KUKA KRL program: MyProgram_201().src

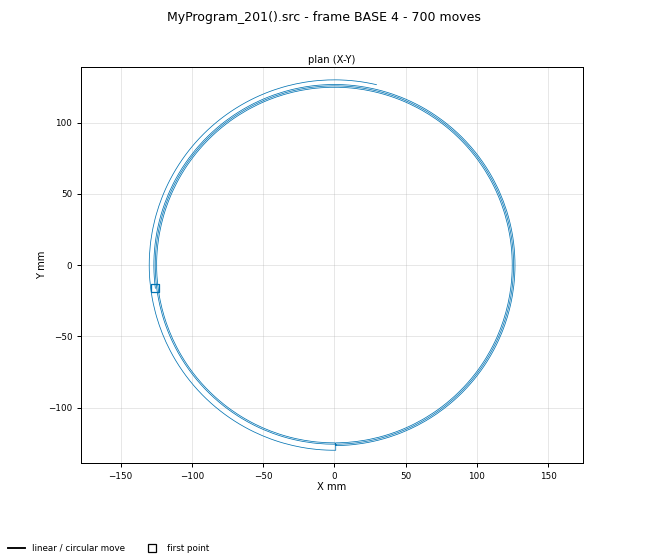
[picture p0: tool path of MyProgram_201().src in frame BASE 4, 700 of 700 moves have a stored position in this frame; points joined in program order, loops and branches not executed]
&ACCESS RVP
&REL 1
&PARAM TEMPLATE = C:\KRC\Roboter\Template\vorgabe
&PARAM EDITMASK = *
DEF MyProgram_201()
; ---- Setting reference (Base) ----
$BASE = BASE_DATA[4]

; --------------------------
; ---- Setting tool (TCP) ----
$TOOL = TOOL_DATA[3]
; --------------------------

$VEL.CP = VEL_APROX_PRINT
Startdeposition()
$VEL.CP = VEL_PRINT
LIN {X -125.6198,Y -16.3,Z 144,A -176.0579,B 23.3517,C -1.2096,E1 23.2223,E2 262.9437} C_DIS
LIN {X -126.0896,Y -12.1409,Z 144,A -177.9619,B 23.3515,C -1.2152,E1 23.2217,E2 264.8457} C_DIS
LIN {X -126.3878,Y -8.5224,Z 144,A -179.6727,B 23.3514,C -1.2176,E1 23.2214,E2 266.5617} C_DIS
LIN {X -126.5802,Y -4.8461,Z 144,A 178.7289,B 23.351,C -1.2257,E1 23.2212,E2 268.1497} C_DIS
LIN {X -126.6703,Y -1.0023,Z 144,A 177.0039,B 23.3506,C -1.2319,E1 23.2211,E2 269.8702} C_DIS
LIN {X -126.6432,Y 2.8281,Z 144,A 175.1115,B 23.3507,C -1.2309,E1 23.2211,E2 271.7776} C_DIS
LIN {X -126.4965,Y 6.6909,Z 144,A 173.3723,B 23.3504,C -1.2369,E1 23.2214,E2 273.5127} C_DIS
LIN {X -126.2226,Y 10.6706,Z 144,A 171.6302,B 23.35,C -1.2454,E1 23.2218,E2 275.2447} C_DIS
LIN {X -125.8208,Y 14.6708,Z 144,A 169.7416,B 23.3498,C -1.2483,E1 23.2223,E2 277.138} C_DIS
LIN {X -125.28,Y 18.7432,Z 144,A 167.8361,B 23.3496,C -1.2523,E1 23.2231,E2 279.0456} C_DIS
LIN {X -124.6746,Y 22.4103,Z 144,A 166.2415,B 23.3492,C -1.2614,E1 23.2238,E2 280.6274} C_DIS
LIN {X -123.8824,Y 26.4422,Z 144,A 164.0896,B 23.3495,C -1.2551,E1 23.2251,E2 282.809} C_DIS
LIN {X -122.8112,Y 31.0384,Z 144,A 162.2249,B 23.3486,C -1.2732,E1 23.2263,E2 284.6396} C_DIS
LIN {X -121.8435,Y 34.6469,Z 144,A 159.9894,B 23.3494,C -1.2558,E1 23.228,E2 286.9331} C_DIS
LIN {X -120.6189,Y 38.6913,Z 144,A 158.5603,B 23.3481,C -1.2819,E1 23.2291,E2 288.305} C_DIS
LIN {X -119.0709,Y 43.2217,Z 144,A 156.4748,B 23.3476,C -1.2919,E1 23.231,E2 290.3777} C_DIS
LIN {X -117.9603,Y 46.1668,Z 144,A 155.028,B 23.3474,C -1.2954,E1 23.2325,E2 291.8245} C_DIS
LIN {X -116.7964,Y 49.0362,Z 144,A 153.2106,B 23.3481,C -1.2823,E1 23.2345,E2 293.686} C_DIS
LIN {X -115.419,Y 52.1955,Z 144,A 151.7283,B 23.3477,C -1.2902,E1 23.2362,E2 295.1571} C_DIS
LIN {X -113.1115,Y 57.0256,Z 144,A 149.2606,B 23.3474,C -1.2954,E1 23.2392,E2 297.6257} C_DIS
LIN {X -111.6267,Y 59.8811,Z 144,A 147.8797,B 23.347,C -1.3028,E1 23.241,E2 298.9958} C_DIS
LIN {X -109.2886,Y 64.0498,Z 144,A 145.8278,B 23.3464,C -1.3137,E1 23.2439,E2 301.0317} C_DIS
LIN {X -106.917,Y 67.9358,Z 144,A 143.7293,B 23.3462,C -1.3179,E1 23.247,E2 303.1311} C_DIS
LIN {X -104.5298,Y 71.5536,Z 144,A 141.7868,B 23.3459,C -1.3241,E1 23.25,E2 305.0683} C_DIS
LIN {X -102.0291,Y 75.0763,Z 144,A 139.8415,B 23.3456,C -1.3298,E1 23.2531,E2 307.0093} C_DIS
LIN {X -97.7758,Y 80.538,Z 144,A 136.8601,B 23.3448,C -1.3444,E1 23.2583,E2 309.9688} C_DIS
LIN {X -95.6486,Y 83.0531,Z 144,A 135.1365,B 23.3451,C -1.3384,E1 23.2614,E2 311.7162} C_DIS
LIN {X -91.6576,Y 87.4372,Z 144,A 132.8632,B 23.3438,C -1.3624,E1 23.2656,E2 313.9395} C_DIS
LIN {X -88.5294,Y 90.6034,Z 144,A 130.4673,B 23.3444,C -1.351,E1 23.2704,E2 316.3752} C_DIS
LIN {X -85.4652,Y 93.4997,Z 144,A 128.2304,B 23.3449,C -1.3415,E1 23.2751,E2 318.646} C_DIS
LIN {X -82.7854,Y 95.88,Z 144,A 126.8175,B 23.3443,C -1.354,E1 23.278,E2 320.0333} C_DIS
LIN {X -79.5981,Y 98.542,Z 144,A 125.0127,B 23.3439,C -1.3612,E1 23.2819,E2 321.8271} C_DIS
LIN {X -76.158,Y 101.2243,Z 144,A 123.1143,B 23.3435,C -1.3686,E1 23.2861,E2 323.7143} C_DIS
LIN {X -70.9814,Y 104.9191,Z 144,A 120.1884,B 23.3433,C -1.3722,E1 23.2928,E2 326.6418} C_DIS
LIN {X -67.4074,Y 107.2505,Z 144,A 118.1775,B 23.3433,C -1.3724,E1 23.2975,E2 328.6591} C_DIS
LIN {X -63.7154,Y 109.4843,Z 144,A 116.2997,B 23.3429,C -1.3791,E1 23.302,E2 330.5261} C_DIS
LIN {X -60.2851,Y 111.4101,Z 144,A 114.4465,B 23.3429,C -1.379,E1 23.3065,E2 332.3853} C_DIS
LIN {X -56.9815,Y 113.134,Z 144,A 112.7261,B 23.3429,C -1.3802,E1 23.3108,E2 334.1076} C_DIS
LIN {X -52.7308,Y 115.1763,Z 144,A 110.7397,B 23.3423,C -1.3899,E1 23.3158,E2 336.075} C_DIS
LIN {X -49.6659,Y 116.5317,Z 144,A 109.2183,B 23.3422,C -1.3918,E1 23.3197,E2 337.5953} C_DIS
LIN {X -46.4891,Y 117.8349,Z 144,A 107.0676,B 23.3435,C -1.3681,E1 23.3254,E2 339.8112} C_DIS
LIN {X -42.2554,Y 119.4193,Z 144,A 105.3156,B 23.3426,C -1.3833,E1 23.3299,E2 341.5284} C_DIS
LIN {X -35.1581,Y 121.6966,Z 144,A 102.0862,B 23.3421,C -1.3933,E1 23.3385,E2 344.7386} C_DIS
LIN {X -30.6403,Y 122.9122,Z 144,A 100.1076,B 23.3416,C -1.4014,E1 23.3438,E2 346.6997} C_DIS
LIN {X -27.0358,Y 123.7543,Z 144,A 98.3688,B 23.3416,C -1.4001,E1 23.3485,E2 348.4443} C_DIS
LIN {X -23.779,Y 124.4208,Z 144,A 96.8918,B 23.3416,C -1.4025,E1 23.3526,E2 349.9172} C_DIS
LIN {X -19.8742,Y 125.1049,Z 144,A 94.9819,B 23.3418,C -1.3986,E1 23.3579,E2 351.8388} C_DIS
LIN {X -15.5594,Y 125.7148,Z 144,A 93.0348,B 23.3417,C -1.4008,E1 23.3633,E2 353.7819} C_DIS
LIN {X -11.7071,Y 126.1313,Z 144,A 90.9218,B 23.3425,C -1.3858,E1 23.3692,E2 355.9341} C_DIS
LIN {X -7.8333,Y 126.4304,Z 144,A 89.507,B 23.3416,C -1.4016,E1 23.3731,E2 357.3093} C_DIS
LIN {X -3.5316,Y 126.6237,Z 144,A 87.6883,B 23.3412,C -1.408,E1 23.3781,E2 359.1124} C_DIS
LIN {X 0.2429,Y 126.6735,Z 144,A 85.6174,B 23.3422,C -1.3921,E1 23.384,E2 361.2235} C_DIS
LIN {X 3.5494,Y 126.6232,Z 144,A 84.81,B 23.3404,C -1.4231,E1 23.386,E2 361.9523} C_DIS
LIN {X 5.9066,Y 126.5359,Z 144,A 83.2679,B 23.3416,C -1.4017,E1 23.3905,E2 363.5479} C_DIS
LIN {X 10.1935,Y 126.2629,Z 144,A 81.4048,B 23.3414,C -1.4052,E1 23.3956,E2 365.4013} C_DIS
LIN {X 13.9971,Y 125.8979,Z 144,A 79.6067,B 23.3416,C -1.4018,E1 23.4007,E2 367.2067} C_DIS
LIN {X 18.4024,Y 125.3298,Z 144,A 77.6752,B 23.3414,C -1.4048,E1 23.406,E2 369.1289} C_DIS
LIN {X 22.234,Y 124.7062,Z 144,A 75.9188,B 23.3414,C -1.4041,E1 23.4108,E2 370.8849} C_DIS
LIN {X 26.3969,Y 123.8922,Z 144,A 74.0065,B 23.3415,C -1.4035,E1 23.416,E2 372.7962} C_DIS
LIN {X 29.8566,Y 123.1039,Z 144,A 72.4577,B 23.3415,C -1.4052,E1 23.4202,E2 374.3385} C_DIS
LIN {X 33.465,Y 122.174,Z 144,A 70.6308,B 23.3418,C -1.3976,E1 23.4252,E2 376.1815} C_DIS
LIN {X 37.2836,Y 121.0616,Z 144,A 68.5449,B 23.3427,C -1.3832,E1 23.4309,E2 378.2997} C_DIS
LIN {X 40.9331,Y 119.8781,Z 144,A 67.3255,B 23.3414,C -1.4053,E1 23.4339,E2 379.4609} C_DIS
LIN {X 46.9072,Y 117.6684,Z 144,A 64.503,B 23.3414,C -1.4052,E1 23.4413,E2 382.2771} C_DIS
LIN {X 50.4597,Y 116.1885,Z 144,A 62.6584,B 23.3418,C -1.3985,E1 23.4461,E2 384.1339} C_DIS
LIN {X 53.5436,Y 114.8005,Z 144,A 60.934,B 23.3424,C -1.3876,E1 23.4505,E2 385.8809} C_DIS
LIN {X 58.0942,Y 112.5675,Z 144,A 58.8505,B 23.342,C -1.3944,E1 23.4557,E2 387.9413} C_DIS
LIN {X 60.6229,Y 111.2261,Z 144,A 57.3893,B 23.3426,C -1.3849,E1 23.4593,E2 389.4219} C_DIS
LIN {X 63.5642,Y 109.5718,Z 144,A 55.9184,B 23.3426,C -1.3852,E1 23.4628,E2 390.8872} C_DIS
LIN {X 67.2338,Y 107.3598,Z 144,A 53.9488,B 23.3428,C -1.3808,E1 23.4675,E2 392.8613} C_DIS
LIN {X 70.8573,Y 105.0027,Z 144,A 51.8125,B 23.3434,C -1.3691,E1 23.4726,E2 395.0192} C_DIS
LIN {X 73.5099,Y 103.1635,Z 144,A 50.8381,B 23.3423,C -1.3894,E1 23.4747,E2 395.939} C_DIS
LIN {X 76.0074,Y 101.338,Z 144,A 49.1263,B 23.3433,C -1.3722,E1 23.4786,E2 397.6875} C_DIS
LIN {X 79.7456,Y 98.423,Z 144,A 47.0444,B 23.3433,C -1.3711,E1 23.4831,E2 399.7637} C_DIS
LIN {X 83.033,Y 95.6661,Z 144,A 45.111,B 23.3435,C -1.3676,E1 23.4872,E2 401.6977} C_DIS
LIN {X 86.1377,Y 92.8802,Z 144,A 43.2356,B 23.3437,C -1.3643,E1 23.4911,E2 403.5732} C_DIS
LIN {X 89.0952,Y 90.0471,Z 144,A 41.3667,B 23.344,C -1.3596,E1 23.4949,E2 405.4457} C_DIS
LIN {X 92.215,Y 86.8491,Z 144,A 39.2479,B 23.3445,C -1.3505,E1 23.499,E2 407.5774} C_DIS
LIN {X 95.66,Y 83.04,Z 144,A 37.0516,B 23.3445,C -1.3512,E1 23.503,E2 409.7614} C_DIS
LIN {X 98.5681,Y 79.5657,Z 144,A 34.8905,B 23.345,C -1.341,E1 23.5069,E2 411.9373} C_DIS
LIN {X 100.9397,Y 76.5352,Z 144,A 33.2696,B 23.3449,C -1.3424,E1 23.5096,E2 413.5464} C_DIS
LIN {X 103.7767,Y 72.6422,Z 144,A 31.1105,B 23.3451,C -1.3379,E1 23.5131,E2 415.7056} C_DIS
LIN {X 106.2024,Y 69.0465,Z 144,A 29.1812,B 23.3453,C -1.3343,E1 23.5161,E2 417.6334} C_DIS
LIN {X 108.9015,Y 64.7054,Z 144,A 26.6855,B 23.3461,C -1.3194,E1 23.5197,E2 420.1529} C_DIS
LIN {X 111.4774,Y 60.16,Z 144,A 24.4951,B 23.3461,C -1.3212,E1 23.5227,E2 422.3265} C_DIS
LIN {X 113.137,Y 56.9755,Z 144,A 23.0738,B 23.3458,C -1.3264,E1 23.5245,E2 423.7263} C_DIS
LIN {X 114.3455,Y 54.507,Z 144,A 21.7849,B 23.3461,C -1.3207,E1 23.526,E2 425.0222} C_DIS
LIN {X 115.7212,Y 51.5224,Z 144,A 20.2942,B 23.3463,C -1.3163,E1 23.5278,E2 426.5154} C_DIS
LIN {X 118.532,Y 44.6783,Z 144,A 17.2084,B 23.3462,C -1.3191,E1 23.531,E2 429.5757} C_DIS
LIN {X 120.9837,Y 37.5382,Z 144,A 13.7256,B 23.3469,C -1.3054,E1 23.5341,E2 433.0715} C_DIS
LIN {X 122.1821,Y 33.436,Z 144,A 11.5325,B 23.3479,C -1.2869,E1 23.5358,E2 435.2977} C_DIS
LIN {X 123.1385,Y 29.7129,Z 144,A 9.9468,B 23.3477,C -1.2889,E1 23.5369,E2 436.8683} C_DIS
LIN {X 123.9757,Y 26.01,Z 144,A 8.1829,B 23.3481,C -1.2813,E1 23.5379,E2 438.6404} C_DIS
LIN {X 124.6529,Y 22.5315,Z 144,A 6.636,B 23.3483,C -1.279,E1 23.5387,E2 440.1833} C_DIS
LIN {X 125.2127,Y 19.1782,Z 144,A 5.1321,B 23.3484,C -1.2758,E1 23.5394,E2 441.6857} C_DIS
LIN {X 125.7472,Y 15.2874,Z 144,A 3.322,B 23.3488,C -1.2685,E1 23.5401,E2 443.5026} C_DIS
LIN {X 126.1487,Y 11.5259,Z 144,A 1.4148,B 23.3496,C -1.2534,E1 23.5406,E2 445.4354} C_DIS
LIN {X 126.4634,Y 7.2985,Z 144,A -0.699,B 23.3504,C -1.2377,E1 23.541,E2 447.5752} C_DIS
LIN {X 126.6257,Y 3.4602,Z 144,A -2.0172,B 23.3496,C -1.2525,E1 23.541,E2 448.8477} C_DIS
LIN {X 126.6741,Y -0.4435,Z 144,A -4.1027,B 23.3507,C -1.2311,E1 23.541,E2 450.9733} C_DIS
LIN {X 126.6143,Y -3.867,Z 144,A -5.4652,B 23.3505,C -1.2352,E1 23.541,E2 452.3169} C_DIS
LIN {X 126.4545,Y -7.4424,Z 144,A -6.8931,B 23.3503,C -1.2393,E1 23.5408,E2 453.7254} C_DIS
LIN {X 126.205,Y -10.8793,Z 144,A -8.4102,B 23.3504,C -1.2363,E1 23.5404,E2 455.2405} C_DIS
LIN {X 125.8638,Y -14.3081,Z 144,A -10.5466,B 23.3521,C -1.203,E1 23.5397,E2 457.4466} C_DIS
LIN {X 125.2715,Y -18.7982,Z 144,A -11.9025,B 23.3507,C -1.2301,E1 23.5392,E2 458.7259} C_DIS
LIN {X 124.8446,Y -21.4515,Z 144,A -13.3029,B 23.3514,C -1.2172,E1 23.5386,E2 460.15} C_DIS
LIN {X 124.1494,Y -25.1576,Z 144,A -14.8753,B 23.3514,C -1.2182,E1 23.5377,E2 461.7098} C_DIS
LIN {X 123.4731,Y -28.2905,Z 144,A -16.3225,B 23.3515,C -1.2137,E1 23.5369,E2 463.1592} C_DIS
LIN {X 122.6734,Y -31.581,Z 144,A -17.9398,B 23.352,C -1.2046,E1 23.5358,E2 464.7893} C_DIS
LIN {X 121.313,Y -36.4621,Z 144,A -20.3518,B 23.3526,C -1.1914,E1 23.5339,E2 467.2194} C_DIS
LIN {X 119.6559,Y -41.574,Z 144,A -22.5939,B 23.3526,C -1.193,E1 23.5319,E2 469.4439} C_DIS
LIN {X 118.4529,Y -44.8894,Z 144,A -24.0956,B 23.3526,C -1.1926,E1 23.5305,E2 470.9375} C_DIS
LIN {X 117.2414,Y -47.9665,Z 144,A -26.4217,B 23.3547,C -1.1477,E1 23.5279,E2 473.3624} C_DIS
LIN {X 115.0168,Y -53.0757,Z 144,A -28.1096,B 23.3532,C -1.1804,E1 23.5261,E2 474.9584} C_DIS
LIN {X 113.536,Y -56.1738,Z 144,A -29.6697,B 23.3534,C -1.1754,E1 23.5242,E2 476.522} C_DIS
LIN {X 111.7463,Y -59.6594,Z 144,A -31.5581,B 23.3539,C -1.1645,E1 23.5217,E2 478.4272} C_DIS
LIN {X 109.5491,Y -63.6034,Z 144,A -33.578,B 23.3541,C -1.1596,E1 23.5189,E2 480.4481} C_DIS
LIN {X 106.9185,Y -67.933,Z 144,A -35.6562,B 23.354,C -1.1634,E1 23.5159,E2 482.5054} C_DIS
LIN {X 105.1316,Y -70.6674,Z 144,A -37.6491,B 23.3553,C -1.1342,E1 23.5127,E2 484.5607} C_DIS
LIN {X 102.9247,Y -73.8438,Z 144,A -38.9435,B 23.3545,C -1.1514,E1 23.5107,E2 485.8052} C_DIS
LIN {X 100.1435,Y -77.5733,Z 144,A -41.3778,B 23.3555,C -1.1297,E1 23.5065,E2 488.2814} C_DIS
LIN {X 98.0196,Y -80.2405,Z 144,A -43.2162,B 23.3564,C -1.1114,E1 23.5032,E2 490.1566} C_DIS
LIN {X 94.8372,Y -83.9778,Z 144,A -44.5715,B 23.3547,C -1.1474,E1 23.5009,E2 491.415} C_DIS
LIN {X 92.9285,Y -86.0858,Z 144,A -46.7033,B 23.3567,C -1.1034,E1 23.4966,E2 493.6472} C_DIS
LIN {X 89.5202,Y -89.6248,Z 144,A -48.8548,B 23.3568,C -1.1013,E1 23.4924,E2 495.794} C_DIS
LIN {X 86.2046,Y -92.8179,Z 144,A -50.2021,B 23.3554,C -1.1317,E1 23.4898,E2 497.0592} C_DIS
LIN {X 83.859,Y -94.9423,Z 144,A -52.375,B 23.3572,C -1.0928,E1 23.4851,E2 499.3204} C_DIS
LIN {X 80.2421,Y -98.0183,Z 144,A -54.5894,B 23.3575,C -1.0848,E1 23.4803,E2 501.5457} C_DIS
LIN {X 76.2072,Y -101.1872,Z 144,A -56.044,B 23.3559,C -1.1212,E1 23.4773,E2 502.9032} C_DIS
LIN {X 71.3958,Y -104.6377,Z 144,A -59.0041,B 23.3568,C -1.1022,E1 23.4705,E2 505.9001} C_DIS
LIN {X 67.4922,Y -107.197,Z 144,A -61.0279,B 23.3568,C -1.1022,E1 23.4657,E2 507.9165} C_DIS
LIN {X 63.8251,Y -109.4206,Z 144,A -62.9374,B 23.3568,C -1.1001,E1 23.4611,E2 509.825} C_DIS
LIN {X 58.3747,Y -112.4216,Z 144,A -65.6581,B 23.3568,C -1.0997,E1 23.4545,E2 512.5384} C_DIS
LIN {X 55.9472,Y -113.6477,Z 144,A -66.9097,B 23.357,C -1.0967,E1 23.4513,E2 513.7939} C_DIS
LIN {X 52.9996,Y -115.052,Z 144,A -69.3957,B 23.3592,C -1.047,E1 23.4448,E2 516.3982} C_DIS
LIN {X 46.9171,Y -117.6644,Z 144,A -71.3464,B 23.3572,C -1.0915,E1 23.44,E2 518.2319} C_DIS
LIN {X 43.9008,Y -118.8222,Z 144,A -73.6629,B 23.3591,C -1.0495,E1 23.4337,E2 520.6489} C_DIS
LIN {X 38.4967,Y -120.6811,Z 144,A -75.0613,B 23.3568,C -1.1019,E1 23.4303,E2 521.9125} C_DIS
LIN {X 34.3658,Y -121.9221,Z 144,A -77.3662,B 23.3576,C -1.083,E1 23.424,E2 524.2606} C_DIS
LIN {X 31.1656,Y -122.7789,Z 144,A -78.8431,B 23.3576,C -1.0825,E1 23.42,E2 525.7365} C_DIS
LIN {X 27.8817,Y -123.5665,Z 144,A -80.5186,B 23.358,C -1.0741,E1 23.4154,E2 527.4305} C_DIS
LIN {X 23.6583,Y -124.4438,Z 144,A -82.3488,B 23.3578,C -1.0781,E1 23.4104,E2 529.2482} C_DIS
LIN {X 19.6454,Y -125.1403,Z 144,A -84.5124,B 23.3585,C -1.0618,E1 23.4044,E2 531.4506} C_DIS
LIN {X 16.3427,Y -125.6142,Z 144,A -85.6833,B 23.3579,C -1.0765,E1 23.4012,E2 532.5834} C_DIS
LIN {X 13.4015,Y -125.962,Z 144,A -86.9789,B 23.3579,C -1.0778,E1 23.3977,E2 533.8748} C_DIS
LIN {X 9.8751,Y -126.289,Z 144,A -89.1079,B 23.3589,C -1.0527,E1 23.3916,E2 536.0658} C_DIS
LIN {X 5.8614,Y -126.5377,Z 144,A -90.569,B 23.3583,C -1.0684,E1 23.3876,E2 537.4867} C_DIS
LIN {X 0.8935,Y -126.6682,Z 144,A -91.828,B 23.3563,C -1.1136,E1 23.3844,E2 538.6315} C_DIS
Enddeposition()
LIN {X 0.8935,Y -126.6682,Z 144,A -91.828,B 23.3563,C -1.1136,E1 23.3844,E2 538.6315} C_DIS
Startdeposition()
$VEL.CP = VEL_PRINT
LIN {X 1.3973,Y -125.7042,Z 144,A -91.3697,B 22.5452,C -0.9874,E1 22.5695,E2 538.3914} C_DIS
LIN {X 4.7103,Y -125.622,Z 144,A -89.8294,B 22.5452,C -0.9893,E1 22.5738,E2 536.8467} C_DIS
LIN {X 9.6558,Y -125.3397,Z 144,A -87.6305,B 22.5452,C -0.9876,E1 22.5799,E2 534.6534} C_DIS
LIN {X 13.3287,Y -125.0015,Z 144,A -86.0596,B 22.5454,C -0.9836,E1 22.5842,E2 533.0942} C_DIS
LIN {X 17.0917,Y -124.5446,Z 144,A -84.1177,B 22.5449,C -0.9943,E1 22.5897,E2 531.1261} C_DIS
LIN {X 21.777,Y -123.8099,Z 144,A -82.1653,B 22.5453,C -0.9864,E1 22.595,E2 529.1964} C_DIS
LIN {X 25.3135,Y -123.1351,Z 144,A -80.4656,B 22.5451,C -0.9905,E1 22.5996,E2 527.4884} C_DIS
LIN {X 29.4259,Y -122.2173,Z 144,A -78.6487,B 22.5452,C -0.9876,E1 22.6046,E2 525.682} C_DIS
LIN {X 32.6566,Y -121.3943,Z 144,A -77.1248,B 22.5452,C -0.9893,E1 22.6087,E2 524.1561} C_DIS
LIN {X 37.8213,Y -119.8862,Z 144,A -74.5204,B 22.5447,C -0.999,E1 22.6157,E2 521.5317} C_DIS
LIN {X 44.3034,Y -117.6443,Z 144,A -71.5515,B 22.5449,C -0.9958,E1 22.6235,E2 518.578} C_DIS
LIN {X 48.1574,Y -116.1201,Z 144,A -69.8944,B 22.5452,C -0.9878,E1 22.6277,E2 516.9458} C_DIS
LIN {X 50.0092,Y -115.3343,Z 144,A -68.364,B 22.544,C -1.0174,E1 22.6318,E2 515.3426} C_DIS
LIN {X 53.5193,Y -113.7503,Z 144,A -66.9131,B 22.5444,C -1.006,E1 22.6354,E2 513.9255} C_DIS
LIN {X 56.4487,Y -112.3248,Z 144,A -65.3839,B 22.5443,C -1.0105,E1 22.6392,E2 512.3894} C_DIS
LIN {X 60.5754,Y -110.1551,Z 144,A -63.3016,B 22.5442,C -1.0121,E1 22.6443,E2 510.3094} C_DIS
LIN {X 64.4835,Y -107.9133,Z 144,A -61.4039,B 22.5443,C -1.0086,E1 22.6489,E2 508.4273} C_DIS
LIN {X 67.5262,Y -106.0362,Z 144,A -59.7903,B 22.5443,C -1.0109,E1 22.6527,E2 506.8135} C_DIS
LIN {X 70.7564,Y -103.9088,Z 144,A -58.0963,B 22.5443,C -1.0112,E1 22.6566,E2 505.1252} C_DIS
LIN {X 73.8837,Y -101.7084,Z 144,A -56.2124,B 22.5438,C -1.0213,E1 22.6609,E2 503.2224} C_DIS
LIN {X 77.115,Y -99.2807,Z 144,A -54.3822,B 22.5436,C -1.0247,E1 22.665,E2 501.391} C_DIS
LIN {X 79.4373,Y -97.4326,Z 144,A -53.0769,B 22.5436,C -1.0254,E1 22.6678,E2 500.0892} C_DIS
LIN {X 83.6912,Y -93.804,Z 144,A -50.6755,B 22.5436,C -1.0243,E1 22.6729,E2 497.7013} C_DIS
LIN {X 87.0109,Y -90.732,Z 144,A -48.3133,B 22.5428,C -1.0432,E1 22.6778,E2 495.3008} C_DIS
LIN {X 90.6624,Y -87.0837,Z 144,A -45.932,B 22.5425,C -1.0503,E1 22.6824,E2 492.9126} C_DIS
LIN {X 93.5791,Y -83.9425,Z 144,A -43.4883,B 22.5413,C -1.0784,E1 22.6871,E2 490.4081} C_DIS
LIN {X 97.0736,Y -79.8764,Z 144,A -41.7141,B 22.5424,C -1.053,E1 22.6901,E2 488.7089} C_DIS
LIN {X 100.5173,Y -75.4965,Z 144,A -39.2558,B 22.5423,C -1.056,E1 22.6943,E2 486.2561} C_DIS
LIN {X 102.6274,Y -72.6018,Z 144,A -37.53,B 22.5419,C -1.0648,E1 22.6972,E2 484.5167} C_DIS
LIN {X 104.4261,Y -69.9902,Z 144,A -36.0169,B 22.5416,C -1.0721,E1 22.6995,E2 482.9932} C_DIS
LIN {X 106.5615,Y -66.6943,Z 144,A -34.3365,B 22.5416,C -1.0719,E1 22.702,E2 481.3226} C_DIS
LIN {X 108.8374,Y -62.9111,Z 144,A -32.4123,B 22.5415,C -1.0735,E1 22.7048,E2 479.4054} C_DIS
LIN {X 110.8877,Y -59.2233,Z 144,A -30.3838,B 22.541,C -1.0841,E1 22.7075,E2 477.3613} C_DIS
LIN {X 112.6381,Y -55.8176,Z 144,A -29.0173,B 22.5416,C -1.0714,E1 22.7092,E2 476.036} C_DIS
LIN {X 113.7558,Y -53.5079,Z 144,A -27.6617,B 22.541,C -1.0837,E1 22.7108,E2 474.6567} C_DIS
LIN {X 115.4559,Y -49.7279,Z 144,A -25.7582,B 22.5407,C -1.0901,E1 22.713,E2 472.7483} C_DIS
LIN {X 116.9827,Y -46.0242,Z 144,A -23.872,B 22.5403,C -1.0985,E1 22.7149,E2 470.8519} C_DIS
LIN {X 118.0398,Y -43.243,Z 144,A -22.5259,B 22.5402,C -1.1022,E1 22.7163,E2 469.5047} C_DIS
LIN {X 119.5913,Y -38.7445,Z 144,A -20.5598,B 22.5403,C -1.0993,E1 22.718,E2 467.5584} C_DIS
LIN {X 121.2999,Y -33.0105,Z 144,A -17.6404,B 22.5395,C -1.117,E1 22.7203,E2 464.612} C_DIS
LIN {X 122.25,Y -29.2905,Z 144,A -16.0088,B 22.5395,C -1.117,E1 22.7214,E2 462.9912} C_DIS
LIN {X 123.0731,Y -25.6183,Z 144,A -14.3435,B 22.5393,C -1.12,E1 22.7224,E2 461.3287} C_DIS
LIN {X 123.7616,Y -22.0466,Z 144,A -12.6352,B 22.539,C -1.1277,E1 22.7232,E2 459.6117} C_DIS
LIN {X 124.4349,Y -17.8596,Z 144,A -10.6377,B 22.5385,C -1.137,E1 22.7241,E2 457.6034} C_DIS
LIN {X 124.996,Y -13.3799,Z 144,A -8.7163,B 22.5385,C -1.137,E1 22.7247,E2 455.6943} C_DIS
LIN {X 125.3442,Y -9.5941,Z 144,A -7.1161,B 22.5385,C -1.1364,E1 22.7251,E2 454.1066} C_DIS
LIN {X 125.5162,Y -7.0136,Z 144,A -5.6321,B 22.5377,C -1.1547,E1 22.7253,E2 452.5851} C_DIS
LIN {X 125.6659,Y -3.337,Z 144,A -4.1352,B 22.5378,C -1.1515,E1 22.7255,E2 451.1064} C_DIS
LIN {X 125.7109,Y 0.4944,Z 144,A -2.2888,B 22.5373,C -1.1618,E1 22.7255,E2 449.2455} C_DIS
LIN {X 125.6122,Y 4.9598,Z 144,A -0.3445,B 22.5373,C -1.164,E1 22.7253,E2 447.3085} C_DIS
LIN {X 125.3828,Y 9.0647,Z 144,A 1.5442,B 22.5369,C -1.1707,E1 22.725,E2 445.415} C_DIS
LIN {X 125.0498,Y 12.8794,Z 144,A 3.3043,B 22.5366,C -1.177,E1 22.7245,E2 443.6504} C_DIS
LIN {X 124.5826,Y 16.8046,Z 144,A 5.0302,B 22.5365,C -1.1791,E1 22.7239,E2 441.9305} C_DIS
LIN {X 124.0343,Y 20.4578,Z 144,A 6.6901,B 22.5363,C -1.1833,E1 22.7232,E2 440.2707} C_DIS
LIN {X 123.3637,Y 24.1809,Z 144,A 8.4722,B 22.5359,C -1.1914,E1 22.7222,E2 438.4793} C_DIS
LIN {X 122.6818,Y 27.4311,Z 144,A 9.9685,B 22.5357,C -1.1952,E1 22.7214,E2 436.9827} C_DIS
LIN {X 121.8425,Y 30.9412,Z 144,A 11.5191,B 22.5357,C -1.1959,E1 22.7203,E2 435.4405} C_DIS
LIN {X 120.8108,Y 34.7569,Z 144,A 13.3945,B 22.5352,C -1.2048,E1 22.7189,E2 433.554} C_DIS
LIN {X 119.1746,Y 40.0056,Z 144,A 15.8059,B 22.535,C -1.2079,E1 22.7169,E2 431.1499} C_DIS
LIN {X 117.9546,Y 43.4749,Z 144,A 17.5608,B 22.5346,C -1.2165,E1 22.7152,E2 429.3837} C_DIS
LIN {X 116.6595,Y 46.8349,Z 144,A 19.4072,B 22.5339,C -1.231,E1 22.7133,E2 427.5112} C_DIS
LIN {X 115.4102,Y 49.8337,Z 144,A 20.5484,B 22.5345,C -1.2193,E1 22.712,E2 426.4074} C_DIS
LIN {X 113.8888,Y 53.2213,Z 144,A 22.2347,B 22.5342,C -1.2238,E1 22.7101,E2 424.7197} C_DIS
LIN {X 112.4489,Y 56.2012,Z 144,A 23.6966,B 22.5342,C -1.2258,E1 22.7083,E2 423.2613} C_DIS
LIN {X 110.4675,Y 60.003,Z 144,A 25.6015,B 22.534,C -1.2289,E1 22.7058,E2 421.3597} C_DIS
LIN {X 106.7236,Y 66.4338,Z 144,A 29.1203,B 22.5332,C -1.2438,E1 22.7008,E2 417.8224} C_DIS
LIN {X 104.517,Y 69.854,Z 144,A 30.973,B 22.5329,C -1.2485,E1 22.6979,E2 415.968} C_DIS
LIN {X 102.3735,Y 72.9595,Z 144,A 32.854,B 22.5323,C -1.2604,E1 22.6949,E2 414.0665} C_DIS
LIN {X 99.8538,Y 76.3714,Z 144,A 35.3234,B 22.5307,C -1.2902,E1 22.6906,E2 411.5328} C_DIS
LIN {X 96.3505,Y 80.7463,Z 144,A 37.1616,B 22.5322,C -1.2627,E1 22.6874,E2 409.7753} C_DIS
LIN {X 93.4225,Y 84.1172,Z 144,A 39.1811,B 22.532,C -1.2667,E1 22.6837,E2 407.7558} C_DIS
LIN {X 90.4829,Y 87.2713,Z 144,A 41.153,B 22.5317,C -1.2713,E1 22.6799,E2 405.7814} C_DIS
LIN {X 87.5036,Y 90.258,Z 144,A 43.0584,B 22.5316,C -1.2746,E1 22.6761,E2 403.8765} C_DIS
LIN {X 84.1876,Y 93.3594,Z 144,A 45.1451,B 22.5313,C -1.2796,E1 22.6718,E2 401.7863} C_DIS
LIN {X 80.894,Y 96.2265,Z 144,A 47.0415,B 22.5313,C -1.2792,E1 22.6678,E2 399.8992} C_DIS
LIN {X 77.7947,Y 98.7491,Z 144,A 48.7644,B 22.5313,C -1.2781,E1 22.6641,E2 398.1865} C_DIS
LIN {X 74.6266,Y 101.1648,Z 144,A 50.59,B 22.5312,C -1.2818,E1 22.66,E2 396.3587} C_DIS
LIN {X 68.4588,Y 105.4361,Z 144,A 54.0629,B 22.5307,C -1.2898,E1 22.652,E2 392.878} C_DIS
LIN {X 65.0458,Y 107.5752,Z 144,A 55.9453,B 22.5305,C -1.2948,E1 22.6475,E2 390.9895} C_DIS
LIN {X 61.7684,Y 109.4901,Z 144,A 57.9194,B 22.5297,C -1.3083,E1 22.6426,E2 388.9868} C_DIS
LIN {X 58.9101,Y 111.053,Z 144,A 58.9352,B 22.5308,C -1.2891,E1 22.6403,E2 388.0241} C_DIS
LIN {X 53.407,Y 113.8029,Z 144,A 61.8058,B 22.5304,C -1.2956,E1 22.6331,E2 385.1453} C_DIS
LIN {X 50.1312,Y 115.2816,Z 144,A 63.447,B 22.5304,C -1.2976,E1 22.6289,E2 383.5033} C_DIS
LIN {X 47.4059,Y 116.4293,Z 144,A 64.6842,B 22.5305,C -1.2941,E1 22.6257,E2 382.2785} C_DIS
LIN {X 45.0897,Y 117.346,Z 144,A 66.1802,B 22.5296,C -1.3114,E1 22.6217,E2 380.7413} C_DIS
LIN {X 40.9801,Y 118.8428,Z 144,A 67.9313,B 22.5301,C -1.3024,E1 22.6172,E2 379.0176} C_DIS
LIN {X 38.2253,Y 119.7571,Z 144,A 69.4464,B 22.5295,C -1.312,E1 22.6131,E2 377.4806} C_DIS
LIN {X 33.614,Y 121.1326,Z 144,A 71.5799,B 22.5295,C -1.3109,E1 22.6074,E2 375.3539} C_DIS
LIN {X 29.5738,Y 122.1817,Z 144,A 73.3621,B 22.5298,C -1.3068,E1 22.6026,E2 373.5856} C_DIS
LIN {X 26.7358,Y 122.8341,Z 144,A 74.6078,B 22.53,C -1.3039,E1 22.5992,E2 372.3493} C_DIS
LIN {X 24.26,Y 123.3486,Z 144,A 76.0118,B 22.5293,C -1.3155,E1 22.5953,E2 370.9169} C_DIS
LIN {X 20.2227,Y 124.0736,Z 144,A 77.8245,B 22.5294,C -1.3137,E1 22.5903,E2 369.1112} C_DIS
LIN {X 16.6715,Y 124.6001,Z 144,A 79.4068,B 22.5295,C -1.3117,E1 22.5859,E2 367.5354} C_DIS
LIN {X 12.7934,Y 125.0591,Z 144,A 81.1548,B 22.5295,C -1.3106,E1 22.5811,E2 365.7916} C_DIS
LIN {X 9.6513,Y 125.34,Z 144,A 82.6613,B 22.5295,C -1.3138,E1 22.5769,E2 364.2779} C_DIS
LIN {X 5.8843,Y 125.573,Z 144,A 84.4407,B 22.5293,C -1.3164,E1 22.5719,E2 362.4924} C_DIS
LIN {X 2.548,Y 125.6852,Z 144,A 85.9635,B 22.5293,C -1.3163,E1 22.5677,E2 360.9701} C_DIS
LIN {X -1.588,Y 125.7011,Z 144,A 87.7905,B 22.5294,C -1.3134,E1 22.5626,E2 359.1507} C_DIS
LIN {X -5.8581,Y 125.5743,Z 144,A 89.6412,B 22.5297,C -1.3086,E1 22.5575,E2 357.3121} C_DIS
LIN {X -9.2502,Y 125.3693,Z 144,A 91.2103,B 22.5297,C -1.3089,E1 22.5531,E2 355.7415} C_DIS
LIN {X -12.6393,Y 125.0746,Z 144,A 92.8985,B 22.5294,C -1.3141,E1 22.5483,E2 354.0388} C_DIS
LIN {X -17.0334,Y 124.5526,Z 144,A 94.8862,B 22.5295,C -1.3117,E1 22.5429,E2 352.0558} C_DIS
LIN {X -20.8143,Y 123.9749,Z 144,A 96.5383,B 22.5298,C -1.3066,E1 22.5383,E2 350.4153} C_DIS
LIN {X -24.7961,Y 123.2404,Z 144,A 98.1445,B 22.5305,C -1.295,E1 22.534,E2 348.8375} C_DIS
LIN {X -27.7971,Y 122.5982,Z 144,A 99.7818,B 22.53,C -1.3039,E1 22.5295,E2 347.1745} C_DIS
LIN {X -30.7189,Y 121.8989,Z 144,A 101.5782,B 22.529,C -1.3209,E1 22.5245,E2 345.3309} C_DIS
LIN {X -34.5541,Y 120.8697,Z 144,A 102.8963,B 22.5303,C -1.298,E1 22.5211,E2 344.0704} C_DIS
LIN {X -41.9598,Y 118.5024,Z 144,A 106.5271,B 22.5303,C -1.2975,E1 22.5115,E2 340.4334} C_DIS
LIN {X -45.6938,Y 117.1111,Z 144,A 108.2688,B 22.5306,C -1.292,E1 22.5069,E2 338.7019} C_DIS
LIN {X -48.0993,Y 116.1444,Z 144,A 109.4942,B 22.5306,C -1.2922,E1 22.5037,E2 337.4729} C_DIS
LIN {X -51.1847,Y 114.8175,Z 144,A 110.9613,B 22.5309,C -1.2874,E1 22.5,E2 336.0146} C_DIS
LIN {X -53.5421,Y 113.7394,Z 144,A 112.3507,B 22.5305,C -1.2943,E1 22.4964,E2 334.6033} C_DIS
LIN {X -56.9349,Y 112.0773,Z 144,A 113.9501,B 22.5309,C -1.2864,E1 22.4925,E2 333.0196} C_DIS
LIN {X -59.9517,Y 110.4955,Z 144,A 115.5264,B 22.531,C -1.2848,E1 22.4886,E2 331.4427} C_DIS
LIN {X -62.9409,Y 108.8201,Z 144,A 117.1463,B 22.531,C -1.2845,E1 22.4847,E2 329.8181} C_DIS
LIN {X -66.1966,Y 106.8712,Z 144,A 118.9254,B 22.531,C -1.2835,E1 22.4804,E2 328.0357} C_DIS
LIN {X -69.4711,Y 104.7726,Z 144,A 120.721,B 22.5312,C -1.281,E1 22.4762,E2 326.2399} C_DIS
LIN {X -73.3963,Y 102.0612,Z 144,A 122.9053,B 22.5314,C -1.2771,E1 22.4712,E2 324.0574} C_DIS
LIN {X -76.7078,Y 99.5964,Z 144,A 124.8137,B 22.5316,C -1.2743,E1 22.467,E2 322.1485} C_DIS
LIN {X -80.0002,Y 96.9711,Z 144,A 126.7172,B 22.5318,C -1.2695,E1 22.4629,E2 320.2496} C_DIS
LIN {X -82.7086,Y 94.6714,Z 144,A 128.3509,B 22.532,C -1.2665,E1 22.4594,E2 318.6166} C_DIS
LIN {X -85.9752,Y 91.7158,Z 144,A 130.3928,B 22.5322,C -1.2633,E1 22.4552,E2 316.5739} C_DIS
LIN {X -89.1602,Y 88.6219,Z 144,A 132.3209,B 22.5326,C -1.2546,E1 22.4514,E2 314.6596} C_DIS
LIN {X -91.5259,Y 86.1765,Z 144,A 133.9755,B 22.5326,C -1.255,E1 22.4482,E2 312.9957} C_DIS
LIN {X -94.5489,Y 82.849,Z 144,A 136.0275,B 22.5329,C -1.25,E1 22.4444,E2 310.9466} C_DIS
LIN {X -97.4805,Y 79.3787,Z 144,A 137.983,B 22.5334,C -1.24,E1 22.441,E2 309.0073} C_DIS
LIN {X -100.2604,Y 75.8369,Z 144,A 140.1506,B 22.5334,C -1.2392,E1 22.4372,E2 306.83} C_DIS
LIN {X -102.7076,Y 72.4882,Z 144,A 142.0685,B 22.5336,C -1.2353,E1 22.4341,E2 304.9121} C_DIS
LIN {X -105.2217,Y 68.7891,Z 144,A 144.1516,B 22.5338,C -1.2314,E1 22.4309,E2 302.8273} C_DIS
LIN {X -107.4248,Y 65.2946,Z 144,A 145.988,B 22.5342,C -1.2242,E1 22.4282,E2 300.9993} C_DIS
LIN {X -109.347,Y 62.0218,Z 144,A 147.5096,B 22.5349,C -1.2108,E1 22.4261,E2 299.504} C_DIS
LIN {X -111.9896,Y 57.1071,Z 144,A 150.2199,B 22.5349,C -1.2102,E1 22.4226,E2 296.7793} C_DIS
LIN {X -113.591,Y 53.8527,Z 144,A 152.5902,B 22.5337,C -1.2345,E1 22.4196,E2 294.3307} C_DIS
LIN {X -115.73,Y 49.0914,Z 144,A 154.2621,B 22.5355,C -1.1984,E1 22.4179,E2 292.743} C_DIS
LIN {X -116.8988,Y 46.2401,Z 144,A 155.8427,B 22.5354,C -1.2013,E1 22.4162,E2 291.145} C_DIS
LIN {X -118.2627,Y 42.6247,Z 144,A 157.535,B 22.5358,C -1.1931,E1 22.4146,E2 289.4634} C_DIS
LIN {X -119.7087,Y 38.377,Z 144,A 159.634,B 22.536,C -1.189,E1 22.4127,E2 287.3618} C_DIS
LIN {X -120.9621,Y 34.2238,Z 144,A 161.539,B 22.5365,C -1.1798,E1 22.4113,E2 285.4684} C_DIS
LIN {X -121.7696,Y 31.2286,Z 144,A 162.784,B 22.537,C -1.1686,E1 22.4104,E2 284.2449} C_DIS
LIN {X -122.4845,Y 28.295,Z 144,A 164.1298,B 22.5373,C -1.163,E1 22.4095,E2 282.9049} C_DIS
LIN {X -123.043,Y 25.7663,Z 144,A 165.8093,B 22.5365,C -1.1794,E1 22.4085,E2 281.1712} C_DIS
LIN {X -123.9653,Y 20.8718,Z 144,A 167.7007,B 22.5376,C -1.1569,E1 22.4076,E2 279.3263} C_DIS
LIN {X -124.4315,Y 17.8833,Z 144,A 169.2086,B 22.5376,C -1.1577,E1 22.407,E2 277.8062} C_DIS
LIN {X -124.946,Y 13.8445,Z 144,A 171.0221,B 22.5379,C -1.15,E1 22.4064,E2 276.0007} C_DIS
LIN {X -125.2603,Y 10.6244,Z 144,A 172.563,B 22.538,C -1.148,E1 22.406,E2 274.4548} C_DIS
LIN {X -125.5343,Y 6.6543,Z 144,A 174.4112,B 22.5382,C -1.1435,E1 22.4057,E2 272.6057} C_DIS
LIN {X -125.6838,Y 2.6278,Z 144,A 176.2903,B 22.5384,C -1.1394,E1 22.4055,E2 270.725} C_DIS
LIN {X -125.7065,Y -1.1296,Z 144,A 178.0855,B 22.5385,C -1.1372,E1 22.4055,E2 268.9232} C_DIS
LIN {X -125.6053,Y -5.137,Z 144,A 179.8881,B 22.5389,C -1.1304,E1 22.4057,E2 267.1263} C_DIS
LIN {X -125.413,Y -8.6522,Z 144,A -178.6267,B 22.5393,C -1.1204,E1 22.406,E2 265.6572} C_DIS
LIN {X -125.1003,Y -12.3711,Z 144,A -176.7514,B 22.5393,C -1.1221,E1 22.4064,E2 263.7649} C_DIS
LIN {X -124.6415,Y -16.3554,Z 144,A -175.0218,B 22.5397,C -1.1123,E1 22.407,E2 262.0493} C_DIS
LIN {X -124.0525,Y -20.3488,Z 144,A -173.2265,B 22.5401,C -1.1048,E1 22.4078,E2 260.2619} C_DIS
LIN {X -123.4772,Y -23.5874,Z 144,A -171.8662,B 22.5405,C -1.0945,E1 22.4085,E2 258.9196} C_DIS
LIN {X -122.4488,Y -28.4512,Z 144,A -169.2579,B 22.5402,C -1.1013,E1 22.41,E2 256.276} C_DIS
LIN {X -120.6353,Y -35.3564,Z 144,A -166.1216,B 22.5409,C -1.0866,E1 22.4123,E2 253.1579} C_DIS
LIN {X -119.435,Y -39.2235,Z 144,A -164.1564,B 22.5409,C -1.086,E1 22.414,E2 251.1818} C_DIS
LIN {X -118.4461,Y -42.1159,Z 144,A -162.796,B 22.5412,C -1.0805,E1 22.4153,E2 249.8271} C_DIS
LIN {X -117.2159,Y -45.4243,Z 144,A -161.2592,B 22.5415,C -1.0729,E1 22.4168,E2 248.3005} C_DIS
LIN {X -116.0214,Y -48.3937,Z 144,A -159.7551,B 22.5416,C -1.0705,E1 22.4184,E2 246.7933} C_DIS
LIN {X -114.6413,Y -51.5787,Z 144,A -158.2161,B 22.5419,C -1.0642,E1 22.4201,E2 245.2613} C_DIS
LIN {X -113.3524,Y -54.3523,Z 144,A -156.7544,B 22.5419,C -1.0631,E1 22.4218,E2 243.7936} C_DIS
LIN {X -111.5604,Y -57.9438,Z 144,A -154.8529,B 22.5421,C -1.0609,E1 22.4243,E2 241.8863} C_DIS
LIN {X -109.5033,Y -61.745,Z 144,A -152.8502,B 22.5422,C -1.0569,E1 22.427,E2 239.8822} C_DIS
LIN {X -107.3306,Y -65.4494,Z 144,A -150.8548,B 22.5424,C -1.0533,E1 22.4298,E2 237.8848} C_DIS
LIN {X -104.7434,Y -69.5148,Z 144,A -148.619,B 22.5426,C -1.0493,E1 22.4332,E2 235.6469} C_DIS
LIN {X -102.1315,Y -73.2979,Z 144,A -146.542,B 22.5428,C -1.0433,E1 22.4366,E2 233.5743} C_DIS
LIN {X -99.4314,Y -76.9207,Z 144,A -144.4475,B 22.543,C -1.0397,E1 22.4401,E2 231.4778} C_DIS
LIN {X -96.5398,Y -80.5207,Z 144,A -142.3317,B 22.5432,C -1.0352,E1 22.4439,E2 229.3628} C_DIS
LIN {X -93.5469,Y -83.9784,Z 144,A -140.3033,B 22.5435,C -1.0282,E1 22.4476,E2 227.3426} C_DIS
LIN {X -90.6491,Y -87.0989,Z 144,A -138.3121,B 22.5435,C -1.026,E1 22.4514,E2 225.3474} C_DIS
LIN {X -87.7943,Y -89.9757,Z 144,A -136.4441,B 22.5437,C -1.023,E1 22.4551,E2 223.4785} C_DIS
LIN {X -84.662,Y -92.9289,Z 144,A -134.4788,B 22.5439,C -1.0191,E1 22.4591,E2 221.5143} C_DIS
LIN {X -81.4152,Y -95.7859,Z 144,A -132.702,B 22.5444,C -1.0071,E1 22.4628,E2 219.7612} C_DIS
LIN {X -78.1,Y -98.508,Z 144,A -130.6301,B 22.5444,C -1.0084,E1 22.4674,E2 217.6772} C_DIS
LIN {X -74.8635,Y -100.9896,Z 144,A -128.2574,B 22.5435,C -1.027,E1 22.4728,E2 215.2463} C_DIS
LIN {X -71.3984,Y -103.4686,Z 144,A -126.7074,B 22.5444,C -1.007,E1 22.4763,E2 213.7426} C_DIS
LIN {X -67.7176,Y -105.9137,Z 144,A -124.8621,B 22.5448,C -0.9967,E1 22.4805,E2 211.9177} C_DIS
LIN {X -64.8026,Y -107.7223,Z 144,A -122.9919,B 22.5444,C -1.0074,E1 22.4851,E2 210.0129} C_DIS
LIN {X -60.6058,Y -110.1382,Z 144,A -121.1441,B 22.5452,C -0.989,E1 22.4895,E2 208.2073} C_DIS
LIN {X -56.2275,Y -112.4359,Z 144,A -118.666,B 22.5449,C -0.9957,E1 22.4957,E2 205.7041} C_DIS
LIN {X -52.9512,Y -114.0137,Z 144,A -117.0944,B 22.5451,C -0.9901,E1 22.4996,E2 204.1427} C_DIS
LIN {X -49.7493,Y -115.4467,Z 144,A -115.4714,B 22.5451,C -0.9893,E1 22.5038,E2 202.5173} C_DIS
LIN {X -45.6775,Y -117.1175,Z 144,A -113.7812,B 22.5458,C -0.9737,E1 22.5081,E2 200.8637} C_DIS
LIN {X -43.2432,Y -118.0397,Z 144,A -112.1574,B 22.5451,C -0.9915,E1 22.5124,E2 199.1898} C_DIS
LIN {X -38.7562,Y -119.5875,Z 144,A -110.0668,B 22.5453,C -0.9866,E1 22.5179,E2 197.1077} C_DIS
LIN {X -35.5337,Y -120.5834,Z 144,A -108.5905,B 22.5454,C -0.9828,E1 22.5219,E2 195.6383} C_DIS
LIN {X -32.3214,Y -121.4837,Z 144,A -107.0667,B 22.5454,C -0.982,E1 22.526,E2 194.1141} C_DIS
LIN {X -28.4745,Y -122.4435,Z 144,A -105.4069,B 22.5458,C -0.9745,E1 22.5304,E2 192.4712} C_DIS
LIN {X -25.2113,Y -123.1559,Z 144,A -103.7563,B 22.5456,C -0.9794,E1 22.535,E2 190.8055} C_DIS
LIN {X -21.9427,Y -123.7802,Z 144,A -102.2073,B 22.5456,C -0.9803,E1 22.5392,E2 189.2525} C_DIS
LIN {X -17.7249,Y -124.4541,Z 144,A -100.3835,B 22.5458,C -0.9744,E1 22.5442,E2 187.4425} C_DIS
LIN {X -15.3658,Y -124.7683,Z 144,A -99.3374,B 22.5458,C -0.9724,E1 22.5471,E2 186.4005} C_DIS
LIN {X -12.5775,Y -125.0805,Z 144,A -97.7909,B 22.5454,C -0.9841,E1 22.5515,E2 184.8226} C_DIS
LIN {X -8.3106,Y -125.4364,Z 144,A -95.9605,B 22.5456,C -0.9787,E1 22.5566,E2 183.0055} C_DIS
LIN {X -5.8356,Y -125.5755,Z 144,A -94.6305,B 22.5452,C -0.9876,E1 22.5604,E2 181.6518} C_DIS
LIN {X -1.6894,Y -125.6994,Z 144,A -92.8902,B 22.5455,C -0.9812,E1 22.5652,E2 179.9281} C_DIS
LIN {X 0.888,Y -125.7071,Z 144,A -92.1808,B 22.5463,C -0.9608,E1 22.567,E2 179.2719} C_DIS
Enddeposition()
LIN {X 0.888,Y -125.7071,Z 144,A -92.1808,B 22.5463,C -0.9608,E1 22.567,E2 179.2719} C_DIS
Startdeposition()
$VEL.CP = VEL_PRINT
LIN {X 0.2524,Y -124.7479,Z 144,A -92.4528,B 21.6328,C -0.8169,E1 21.6473,E2 179.8151} C_DIS
LIN {X -2.8004,Y -124.7177,Z 144,A -93.8116,B 21.6328,C -0.8185,E1 21.6435,E2 181.1697} C_DIS
LIN {X -5.8687,Y -124.6098,Z 144,A -95.3337,B 21.6329,C -0.8138,E1 21.6392,E2 182.7051} C_DIS
LIN {X -8.918,Y -124.4282,Z 144,A -96.719,B 21.6329,C -0.8145,E1 21.6353,E2 184.0889} C_DIS
LIN {X -11.9747,Y -124.1712,Z 144,A -98.1094,B 21.6329,C -0.8154,E1 21.6315,E2 185.4777} C_DIS
LIN {X -15.2704,Y -123.81,Z 144,A -99.586,B 21.6329,C -0.8176,E1 21.6274,E2 186.9496} C_DIS
LIN {X -18.2991,Y -123.3995,Z 144,A -100.9842,B 21.6328,C -0.8181,E1 21.6235,E2 188.3477} C_DIS
LIN {X -21.0776,Y -122.9548,Z 144,A -102.3448,B 21.6328,C -0.8157,E1 21.6197,E2 189.7162} C_DIS
LIN {X -24.0877,Y -122.4013,Z 144,A -103.7803,B 21.6328,C -0.815,E1 21.6158,E2 191.1554} C_DIS
LIN {X -27.0795,Y -121.7746,Z 144,A -105.1144,B 21.6328,C -0.8186,E1 21.6122,E2 192.4818} C_DIS
LIN {X -30.8178,Y -120.8805,Z 144,A -106.9181,B 21.6328,C -0.818,E1 21.6073,E2 194.29} C_DIS
LIN {X -34.7477,Y -119.8103,Z 144,A -108.7516,B 21.6327,C -0.8208,E1 21.6024,E2 196.1193} C_DIS
LIN {X -38.3606,Y -118.7032,Z 144,A -110.6677,B 21.6329,C -0.8148,E1 21.5972,E2 198.0558} C_DIS
LIN {X -42.0313,Y -117.4532,Z 144,A -112.1555,B 21.6324,C -0.8282,E1 21.5934,E2 199.5105} C_DIS
LIN {X -44.6529,Y -116.4828,Z 144,A -113.554,B 21.6325,C -0.8247,E1 21.5897,E2 200.9218} C_DIS
LIN {X -47.7441,Y -115.2493,Z 144,A -115.0912,B 21.6325,C -0.8259,E1 21.5857,E2 202.4598} C_DIS
LIN {X -50.322,Y -114.1487,Z 144,A -116.3775,B 21.6325,C -0.8273,E1 21.5824,E2 203.7457} C_DIS
LIN {X -53.1051,Y -112.8812,Z 144,A -117.8779,B 21.6325,C -0.8251,E1 21.5786,E2 205.2567} C_DIS
LIN {X -55.6295,Y -111.6573,Z 144,A -119.1842,B 21.6325,C -0.826,E1 21.5753,E2 206.5646} C_DIS
LIN {X -58.8172,Y -110.0129,Z 144,A -120.8764,B 21.6325,C -0.8263,E1 21.5711,E2 208.2614} C_DIS
LIN {X -62.7594,Y -107.8127,Z 144,A -122.7937,B 21.6322,C -0.8354,E1 21.5665,E2 210.1604} C_DIS
LIN {X -65.2277,Y -106.3371,Z 144,A -124.1927,B 21.6322,C -0.8343,E1 21.5631,E2 211.5676} C_DIS
LIN {X -68.0304,Y -104.5663,Z 144,A -125.8027,B 21.6322,C -0.8332,E1 21.5593,E2 213.1868} C_DIS
LIN {X -71.6486,Y -102.1215,Z 144,A -127.7456,B 21.632,C -0.8389,E1 21.5549,E2 215.1216} C_DIS
LIN {X -74.3226,Y -100.192,Z 144,A -129.1995,B 21.6318,C -0.8439,E1 21.5516,E2 216.568} C_DIS
LIN {X -77.3473,Y -97.8763,Z 144,A -131.1281,B 21.632,C -0.84,E1 21.5473,E2 218.5156} C_DIS
LIN {X -80.9006,Y -94.9597,Z 144,A -133.2085,B 21.6318,C -0.8452,E1 21.5429,E2 220.5911} C_DIS
LIN {X -83.9176,Y -92.3044,Z 144,A -135.0595,B 21.6317,C -0.8486,E1 21.539,E2 222.4414} C_DIS
LIN {X -87.1252,Y -89.2834,Z 144,A -137.1298,B 21.6316,C -0.851,E1 21.5348,E2 224.5154} C_DIS
LIN {X -90.3489,Y -86.0196,Z 144,A -139.2549,B 21.6314,C -0.8548,E1 21.5307,E2 226.6408} C_DIS
LIN {X -93.3636,Y -82.7374,Z 144,A -141.3112,B 21.6313,C -0.859,E1 21.5269,E2 228.6965} C_DIS
LIN {X -96.3526,Y -79.2374,Z 144,A -143.4384,B 21.6311,C -0.8634,E1 21.523,E2 230.8232} C_DIS
LIN {X -99.286,Y -75.529,Z 144,A -145.6202,B 21.6309,C -0.8682,E1 21.5193,E2 233.0041} C_DIS
LIN {X -101.8411,Y -72.0462,Z 144,A -147.5137,B 21.6306,C -0.8765,E1 21.5162,E2 234.8855} C_DIS
LIN {X -103.4952,Y -69.6498,Z 144,A -148.8323,B 21.6304,C -0.8806,E1 21.5142,E2 236.2007} C_DIS
LIN {X -105.394,Y -66.7412,Z 144,A -150.4044,B 21.6303,C -0.8856,E1 21.5118,E2 237.7684} C_DIS
LIN {X -107.3381,Y -63.568,Z 144,A -152.2689,B 21.6303,C -0.8841,E1 21.5091,E2 239.6483} C_DIS
LIN {X -109.0083,Y -60.6589,Z 144,A -153.7998,B 21.6301,C -0.8886,E1 21.507,E2 241.1764} C_DIS
LIN {X -110.7313,Y -57.4517,Z 144,A -155.3541,B 21.6298,C -0.8977,E1 21.505,E2 242.7157} C_DIS
LIN {X -112.105,Y -54.722,Z 144,A -156.7717,B 21.6296,C -0.901,E1 21.5032,E2 244.1331} C_DIS
LIN {X -113.3721,Y -52.0448,Z 144,A -158.1603,B 21.6296,C -0.9038,E1 21.5016,E2 245.5231} C_DIS
LIN {X -114.6559,Y -49.1522,Z 144,A -159.5638,B 21.6293,C -0.9098,E1 21.5,E2 246.9192} C_DIS
LIN {X -115.7277,Y -46.5712,Z 144,A -160.9466,B 21.6293,C -0.9098,E1 21.4985,E2 248.3113} C_DIS
LIN {X -116.9316,Y -43.4612,Z 144,A -162.4448,B 21.6291,C -0.9154,E1 21.4971,E2 249.8039} C_DIS
LIN {X -117.877,Y -40.8265,Z 144,A -163.8657,B 21.6291,C -0.9141,E1 21.4957,E2 251.2379} C_DIS
LIN {X -119.301,Y -36.4564,Z 144,A -165.8387,B 21.6287,C -0.9256,E1 21.4941,E2 253.1929} C_DIS
LIN {X -120.1801,Y -33.4453,Z 144,A -167.3468,B 21.6286,C -0.9273,E1 21.4929,E2 254.7064} C_DIS
LIN {X -120.9512,Y -30.5395,Z 144,A -168.7032,B 21.6284,C -0.9325,E1 21.492,E2 256.0582} C_DIS
LIN {X -121.7122,Y -27.3526,Z 144,A -170.1618,B 21.6281,C -0.9388,E1 21.4911,E2 257.5095} C_DIS
LIN {X -122.2999,Y -24.5897,Z 144,A -171.5531,B 21.6281,C -0.9392,E1 21.4903,E2 258.9093} C_DIS
LIN {X -122.8665,Y -21.5829,Z 144,A -172.9593,B 21.6279,C -0.9435,E1 21.4896,E2 260.3135} C_DIS
LIN {X -123.4657,Y -17.8359,Z 144,A -174.7563,B 21.6278,C -0.9469,E1 21.4888,E2 262.1139} C_DIS
LIN {X -123.9605,Y -14.0034,Z 144,A -176.5073,B 21.6275,C -0.9533,E1 21.4882,E2 263.8597} C_DIS
LIN {X -124.2874,Y -10.7037,Z 144,A -177.958,B 21.6272,C -0.9609,E1 21.4878,E2 265.2999} C_DIS
LIN {X -124.5122,Y -7.6551,Z 144,A -179.56,B 21.6273,C -0.9579,E1 21.4875,E2 266.9216} C_DIS
LIN {X -124.6989,Y -3.4773,Z 144,A 178.5669,B 21.627,C -0.9657,E1 21.4873,E2 268.7864} C_DIS
LIN {X -124.7512,Y 0,Z 144,A 176.9955,B 21.6267,C -0.9717,E1 21.4873,E2 270.3526} C_DIS
LIN {X -124.7178,Y 2.7981,Z 144,A 175.6188,B 21.6267,C -0.9724,E1 21.4873,E2 271.7372} C_DIS
LIN {X -124.5975,Y 6.1146,Z 144,A 174.1544,B 21.6264,C -0.9795,E1 21.4875,E2 273.1925} C_DIS
LIN {X -124.3755,Y 9.6396,Z 144,A 172.3482,B 21.6264,C -0.9778,E1 21.4879,E2 275.0163} C_DIS
LIN {X -123.9878,Y 13.7499,Z 144,A 170.6451,B 21.6259,C -0.991,E1 21.4884,E2 276.6952} C_DIS
LIN {X -123.6144,Y 16.7829,Z 144,A 169.2327,B 21.6257,C -0.9952,E1 21.4889,E2 278.1062} C_DIS
LIN {X -123.2062,Y 19.5526,Z 144,A 167.9585,B 21.6255,C -0.9997,E1 21.4894,E2 279.377} C_DIS
LIN {X -122.7289,Y 22.3518,Z 144,A 166.5947,B 21.6255,C -1.0015,E1 21.4901,E2 280.7452} C_DIS
LIN {X -122.0399,Y 25.8519,Z 144,A 165.053,B 21.625,C -1.0103,E1 21.4909,E2 282.2736} C_DIS
LIN {X -121.4301,Y 28.5832,Z 144,A 163.5749,B 21.6252,C -1.0071,E1 21.4919,E2 283.7707} C_DIS
LIN {X -120.6276,Y 31.795,Z 144,A 162.2226,B 21.6247,C -1.0182,E1 21.4928,E2 285.1019} C_DIS
LIN {X -119.8126,Y 34.7399,Z 144,A 160.7157,B 21.6247,C -1.0187,E1 21.4939,E2 286.6179} C_DIS
LIN {X -118.9904,Y 37.4616,Z 144,A 159.3317,B 21.6247,C -1.0197,E1 21.4951,E2 288.0084} C_DIS
LIN {X -117.7586,Y 41.1681,Z 144,A 157.4776,B 21.6245,C -1.023,E1 21.4968,E2 289.866} C_DIS
LIN {X -116.4821,Y 44.6548,Z 144,A 155.7332,B 21.6243,C -1.0267,E1 21.4985,E2 291.6118} C_DIS
LIN {X -114.854,Y 48.6907,Z 144,A 153.7999,B 21.6239,C -1.0351,E1 21.5005,E2 293.5347} C_DIS
LIN {X -113.5271,Y 51.7096,Z 144,A 152.3345,B 21.6236,C -1.0415,E1 21.5022,E2 294.9922} C_DIS
LIN {X -112.1064,Y 54.7192,Z 144,A 150.8971,B 21.6233,C -1.0494,E1 21.5039,E2 296.4171} C_DIS
LIN {X -110.7366,Y 57.4417,Z 144,A 149.28,B 21.6235,C -1.0453,E1 21.506,E2 298.0557} C_DIS
LIN {X -108.6685,Y 61.2653,Z 144,A 147.3341,B 21.6231,C -1.0529,E1 21.5086,E2 299.9928} C_DIS
LIN {X -107.1334,Y 63.9115,Z 144,A 145.8689,B 21.6231,C -1.0546,E1 21.5107,E2 301.4623} C_DIS
LIN {X -104.9029,Y 67.5109,Z 144,A 143.8645,B 21.6229,C -1.0577,E1 21.5137,E2 303.4702} C_DIS
LIN {X -102.8639,Y 70.5781,Z 144,A 142.3729,B 21.6223,C -1.0699,E1 21.5159,E2 304.9371} C_DIS
LIN {X -101.1034,Y 73.0779,Z 144,A 140.8902,B 21.6223,C -1.0707,E1 21.5184,E2 306.4262} C_DIS
LIN {X -99.5146,Y 75.227,Z 144,A 139.5798,B 21.6223,C -1.0708,E1 21.5206,E2 307.7437} C_DIS
LIN {X -96.9904,Y 78.4546,Z 144,A 137.7323,B 21.622,C -1.077,E1 21.5238,E2 309.5846} C_DIS
LIN {X -94.5433,Y 81.3868,Z 144,A 135.9402,B 21.6218,C -1.08,E1 21.527,E2 311.3782} C_DIS
LIN {X -91.8324,Y 84.4337,Z 144,A 133.9744,B 21.6218,C -1.0811,E1 21.5307,E2 313.3513} C_DIS
LIN {X -88.7425,Y 87.6763,Z 144,A 131.8775,B 21.6216,C -1.0845,E1 21.5348,E2 315.4495} C_DIS
LIN {X -85.4623,Y 90.8761,Z 144,A 129.7591,B 21.6214,C -1.0889,E1 21.539,E2 317.5663} C_DIS
LIN {X -82.147,Y 93.8836,Z 144,A 127.8253,B 21.621,C -1.0982,E1 21.543,E2 319.4838} C_DIS
LIN {X -79.2339,Y 96.3554,Z 144,A 126.0585,B 21.6208,C -1.1015,E1 21.5468,E2 321.2495} C_DIS
LIN {X -76.2462,Y 98.736,Z 144,A 124.1891,B 21.6208,C -1.1007,E1 21.5509,E2 323.129} C_DIS
LIN {X -73.2919,Y 100.9482,Z 144,A 122.6253,B 21.6204,C -1.1092,E1 21.5544,E2 324.6762} C_DIS
LIN {X -70.5703,Y 102.8692,Z 144,A 121.0847,B 21.6204,C -1.1118,E1 21.5579,E2 326.216} C_DIS
LIN {X -67.4871,Y 104.9181,Z 144,A 119.2472,B 21.6204,C -1.1097,E1 21.5623,E2 328.0663} C_DIS
LIN {X -64.1345,Y 107.0005,Z 144,A 117.5608,B 21.62,C -1.1178,E1 21.5662,E2 329.7366} C_DIS
LIN {X -61.7204,Y 108.4105,Z 144,A 116.222,B 21.62,C -1.1179,E1 21.5695,E2 331.0799} C_DIS
LIN {X -59.2142,Y 109.7996,Z 144,A 114.8737,B 21.62,C -1.1188,E1 21.5728,E2 332.4302} C_DIS
LIN {X -56.3046,Y 111.3178,Z 144,A 113.3999,B 21.6198,C -1.1226,E1 21.5764,E2 333.8985} C_DIS
LIN {X -53.5596,Y 112.6641,Z 144,A 111.9867,B 21.6197,C -1.1244,E1 21.58,E2 335.311} C_DIS
LIN {X -49.86,Y 114.3499,Z 144,A 110.0267,B 21.6197,C -1.1234,E1 21.585,E2 337.2791} C_DIS
LIN {X -46.5617,Y 115.7315,Z 144,A 108.4579,B 21.6195,C -1.1286,E1 21.589,E2 338.8381} C_DIS
LIN {X -43.4579,Y 116.9329,Z 144,A 106.9958,B 21.6193,C -1.1331,E1 21.5928,E2 340.2913} C_DIS
LIN {X -40.7617,Y 117.8995,Z 144,A 105.6509,B 21.6193,C -1.1336,E1 21.5964,E2 341.6382} C_DIS
LIN {X -37.8914,Y 118.8531,Z 144,A 104.2568,B 21.6192,C -1.135,E1 21.6001,E2 343.0314} C_DIS
LIN {X -34.9883,Y 119.7398,Z 144,A 102.8589,B 21.6191,C -1.1363,E1 21.6038,E2 344.4284} C_DIS
LIN {X -31.9893,Y 120.5758,Z 144,A 101.4323,B 21.6191,C -1.1379,E1 21.6077,E2 345.8534} C_DIS
LIN {X -29.0722,Y 121.3122,Z 144,A 100.0056,B 21.6191,C -1.1373,E1 21.6115,E2 347.2838} C_DIS
LIN {X -25.8354,Y 122.0435,Z 144,A 98.5372,B 21.6189,C -1.1408,E1 21.6155,E2 348.745} C_DIS
LIN {X -23.4811,Y 122.5173,Z 144,A 97.3772,B 21.6189,C -1.1394,E1 21.6187,E2 349.9103} C_DIS
LIN {X -19.8131,Y 123.1658,Z 144,A 95.6782,B 21.6189,C -1.141,E1 21.6234,E2 351.6069} C_DIS
LIN {X -17.038,Y 123.5797,Z 144,A 94.4155,B 21.6188,C -1.1429,E1 21.6269,E2 352.8657} C_DIS
LIN {X -13.7487,Y 123.9879,Z 144,A 92.7541,B 21.619,C -1.1381,E1 21.6315,E2 354.5414} C_DIS
LIN {X -9.4196,Y 124.3916,Z 144,A 90.8117,B 21.6189,C -1.1412,E1 21.6369,E2 356.4765} C_DIS
LIN {X -6.3691,Y 124.5847,Z 144,A 89.4595,B 21.6187,C -1.1437,E1 21.6407,E2 357.8222} C_DIS
LIN {X -3.3157,Y 124.7034,Z 144,A 88.0864,B 21.6187,C -1.1453,E1 21.6445,E2 359.1911} C_DIS
LIN {X -0.2603,Y 124.7479,Z 144,A 86.6834,B 21.6187,C -1.1456,E1 21.6484,E2 360.5934} C_DIS
LIN {X 2.8086,Y 124.7175,Z 144,A 85.1585,B 21.6189,C -1.1411,E1 21.6527,E2 362.1304} C_DIS
LIN {X 5.862,Y 124.6102,Z 144,A 83.776,B 21.6189,C -1.142,E1 21.6565,E2 363.51} C_DIS
LIN {X 8.9233,Y 124.4278,Z 144,A 82.3901,B 21.6188,C -1.1428,E1 21.6604,E2 364.8928} C_DIS
LIN {X 11.9697,Y 124.1717,Z 144,A 81.0025,B 21.6188,C -1.1433,E1 21.6642,E2 366.2781} C_DIS
LIN {X 15.2654,Y 123.8106,Z 144,A 79.5268,B 21.6187,C -1.1449,E1 21.6683,E2 367.7481} C_DIS
LIN {X 18.3091,Y 123.3981,Z 144,A 78.1281,B 21.6187,C -1.145,E1 21.6722,E2 369.1452} C_DIS
LIN {X 21.0762,Y 122.9551,Z 144,A 76.7723,B 21.6188,C -1.1417,E1 21.6759,E2 370.5082} C_DIS
LIN {X 24.0829,Y 122.4022,Z 144,A 75.3413,B 21.6189,C -1.14,E1 21.6799,E2 371.9421} C_DIS
LIN {X 27.0747,Y 121.7757,Z 144,A 74.033,B 21.6187,C -1.1432,E1 21.6834,E2 373.2396} C_DIS
LIN {X 31.7974,Y 120.627,Z 144,A 71.784,B 21.6188,C -1.1412,E1 21.6895,E2 375.4901} C_DIS
LIN {X 35.5282,Y 119.5818,Z 144,A 69.8449,B 21.6192,C -1.1333,E1 21.6948,E2 377.4469} C_DIS
LIN {X 39.1363,Y 118.4493,Z 144,A 68.2135,B 21.6191,C -1.1363,E1 21.6991,E2 379.0666} C_DIS
LIN {X 43.0124,Y 117.0995,Z 144,A 66.3193,B 21.6192,C -1.1341,E1 21.704,E2 380.9619} C_DIS
LIN {X 46.0884,Y 115.9224,Z 144,A 64.8074,B 21.6192,C -1.1327,E1 21.708,E2 382.4739} C_DIS
LIN {X 49.7453,Y 114.3995,Z 144,A 62.9841,B 21.6194,C -1.1305,E1 21.7127,E2 384.2979} C_DIS
LIN {X 52.7478,Y 113.047,Z 144,A 61.4294,B 21.6196,C -1.127,E1 21.7166,E2 385.8576} C_DIS
LIN {X 55.8794,Y 111.5341,Z 144,A 59.9637,B 21.6194,C -1.1305,E1 21.7203,E2 387.3092} C_DIS
LIN {X 58.1907,Y 110.3433,Z 144,A 58.866,B 21.6193,C -1.133,E1 21.723,E2 388.3964} C_DIS
LIN {X 61.2703,Y 108.6656,Z 144,A 57.1345,B 21.6196,C -1.1256,E1 21.7272,E2 390.142} C_DIS
LIN {X 63.9163,Y 107.1305,Z 144,A 55.7751,B 21.6196,C -1.1255,E1 21.7305,E2 391.4969} C_DIS
LIN {X 66.1899,Y 105.7414,Z 144,A 54.4657,B 21.6199,C -1.12,E1 21.7336,E2 392.8163} C_DIS
LIN {X 69.3784,Y 103.6769,Z 144,A 52.8217,B 21.6199,C -1.1215,E1 21.7374,E2 394.4499} C_DIS
LIN {X 71.6566,Y 102.1159,Z 144,A 51.4996,B 21.6201,C -1.117,E1 21.7405,E2 395.7786} C_DIS
LIN {X 74.2503,Y 100.2458,Z 144,A 49.9454,B 21.6204,C -1.1108,E1 21.744,E2 397.3431} C_DIS
LIN {X 77.4542,Y 97.7915,Z 144,A 48.0953,B 21.6205,C -1.1076,E1 21.7481,E2 399.1939} C_DIS
LIN {X 80.9019,Y 94.9586,Z 144,A 46.1655,B 21.6205,C -1.1088,E1 21.7522,E2 401.1117} C_DIS
LIN {X 83.7825,Y 92.4269,Z 144,A 44.2999,B 21.6208,C -1.1008,E1 21.7561,E2 402.9902} C_DIS
LIN {X 87.1229,Y 89.2857,Z 144,A 42.2041,B 21.621,C -1.0969,E1 21.7603,E2 405.0863} C_DIS
LIN {X 90.2557,Y 86.1171,Z 144,A 40.2992,B 21.621,C -1.0986,E1 21.764,E2 406.977} C_DIS
LIN {X 92.8593,Y 83.3031,Z 144,A 38.4726,B 21.6213,C -1.0918,E1 21.7675,E2 408.8125} C_DIS
LIN {X 95.5986,Y 80.1445,Z 144,A 36.5449,B 21.6215,C -1.0871,E1 21.771,E2 410.7428} C_DIS
LIN {X 98.3612,Y 76.7297,Z 144,A 34.4938,B 21.6218,C -1.0808,E1 21.7745,E2 412.7995} C_DIS
LIN {X 100.936,Y 73.3088,Z 144,A 32.6959,B 21.6217,C -1.0833,E1 21.7775,E2 414.5804} C_DIS
LIN {X 102.8684,Y 70.5715,Z 144,A 31.2399,B 21.6217,C -1.0831,E1 21.7798,E2 416.0286} C_DIS
LIN {X 104.4249,Y 68.2483,Z 144,A 29.979,B 21.6218,C -1.0808,E1 21.7818,E2 417.2883} C_DIS
LIN {X 106.067,Y 65.6668,Z 144,A 28.4361,B 21.6223,C -1.0711,E1 21.7841,E2 418.8481} C_DIS
LIN {X 107.792,Y 62.7953,Z 144,A 27.0081,B 21.6223,C -1.0719,E1 21.7861,E2 420.2655} C_DIS
LIN {X 108.9761,Y 60.7171,Z 144,A 25.8578,B 21.6225,C -1.0667,E1 21.7877,E2 421.4229} C_DIS
LIN {X 110.5089,Y 57.8754,Z 144,A 24.3687,B 21.6227,C -1.0624,E1 21.7896,E2 422.9143} C_DIS
LIN {X 112.1086,Y 54.7148,Z 144,A 22.8061,B 21.6227,C -1.0607,E1 21.7916,E2 424.4716} C_DIS
LIN {X 113.416,Y 51.9497,Z 144,A 21.2739,B 21.6232,C -1.0512,E1 21.7934,E2 426.0199} C_DIS
LIN {X 115.1579,Y 47.9629,Z 144,A 19.4096,B 21.6232,C -1.0514,E1 21.7954,E2 427.8716} C_DIS
LIN {X 116.3904,Y 44.8907,Z 144,A 17.8991,B 21.6234,C -1.0474,E1 21.797,E2 429.383} C_DIS
LIN {X 117.6166,Y 41.5776,Z 144,A 16.0769,B 21.624,C -1.0338,E1 21.7987,E2 431.2299} C_DIS
LIN {X 118.8392,Y 37.9348,Z 144,A 14.6236,B 21.6236,C -1.0424,E1 21.8,E2 432.6504} C_DIS
LIN {X 119.7384,Y 34.9932,Z 144,A 13.1346,B 21.6239,C -1.0348,E1 21.8012,E2 434.15} C_DIS
LIN {X 120.6142,Y 31.8455,Z 144,A 11.7197,B 21.6239,C -1.034,E1 21.8022,E2 435.5573} C_DIS
LIN {X 121.2895,Y 29.1664,Z 144,A 10.3346,B 21.6244,C -1.025,E1 21.8031,E2 436.9573} C_DIS
LIN {X 122.043,Y 25.8377,Z 144,A 8.8551,B 21.6244,C -1.0241,E1 21.804,E2 438.4293} C_DIS
LIN {X 122.6404,Y 22.837,Z 144,A 7.4551,B 21.6246,C -1.02,E1 21.8048,E2 439.8307} C_DIS
LIN {X 123.0327,Y 20.6106,Z 144,A 6.3703,B 21.6249,C -1.0147,E1 21.8053,E2 440.9223} C_DIS
LIN {X 123.5791,Y 17.0424,Z 144,A 4.7721,B 21.6249,C -1.0122,E1 21.8059,E2 442.5162} C_DIS
LIN {X 123.9601,Y 14.0076,Z 144,A 3.349,B 21.6252,C -1.0069,E1 21.8064,E2 443.9436} C_DIS
LIN {X 124.2871,Y 10.7069,Z 144,A 1.8461,B 21.6254,C -1.0031,E1 21.8068,E2 445.4464} C_DIS
LIN {X 124.5627,Y 6.8067,Z 144,A -0.0922,B 21.6259,C -0.991,E1 21.8071,E2 447.4037} C_DIS
LIN {X 124.7033,Y 3.3162,Z 144,A -1.5433,B 21.6259,C -0.9928,E1 21.8073,E2 448.8399} C_DIS
LIN {X 124.7512,Y 0.0032,Z 144,A -3.2805,B 21.6265,C -0.9783,E1 21.8073,E2 450.6042} C_DIS
LIN {X 124.6627,Y -4.6003,Z 144,A -5.065,B 21.6261,C -0.9863,E1 21.8072,E2 452.3545} C_DIS
LIN {X 124.5123,Y -7.6536,Z 144,A -6.594,B 21.6265,C -0.9763,E1 21.8069,E2 453.8999} C_DIS
LIN {X 124.1719,Y -11.9674,Z 144,A -8.532,B 21.6267,C -0.9721,E1 21.8065,E2 455.8355} C_DIS
LIN {X 123.8109,Y -15.2636,Z 144,A -9.9963,B 21.6268,C -0.9699,E1 21.806,E2 457.2957} C_DIS
LIN {X 123.398,Y -18.3094,Z 144,A -11.391,B 21.627,C -0.9662,E1 21.8054,E2 458.6908} C_DIS
LIN {X 122.9556,Y -21.073,Z 144,A -12.7319,B 21.6272,C -0.9596,E1 21.8048,E2 460.0402} C_DIS
LIN {X 122.4024,Y -24.0821,Z 144,A -14.155,B 21.6275,C -0.9543,E1 21.8041,E2 461.4677} C_DIS
LIN {X 121.7758,Y -27.0738,Z 144,A -15.478,B 21.6275,C -0.9535,E1 21.8033,E2 462.7838} C_DIS
LIN {X 121.0111,Y -30.3034,Z 144,A -16.9879,B 21.6277,C -0.9494,E1 21.8023,E2 464.2945} C_DIS
LIN {X 120.3015,Y -33.0112,Z 144,A -18.3523,B 21.628,C -0.9419,E1 21.8013,E2 465.6701} C_DIS
LIN {X 119.3725,Y -36.2231,Z 144,A -19.7844,B 21.628,C -0.9417,E1 21.8002,E2 467.0929} C_DIS
LIN {X 118.4518,Y -39.1287,Z 144,A -21.1782,B 21.6282,C -0.9377,E1 21.799,E2 468.4883} C_DIS
LIN {X 117.4532,Y -42.0313,Z 144,A -22.4837,B 21.6282,C -0.938,E1 21.7978,E2 469.7844} C_DIS
LIN {X 116.655,Y -44.1998,Z 144,A -23.7127,B 21.6286,C -0.9273,E1 21.7966,E2 471.0342} C_DIS
LIN {X 115.2539,Y -47.7332,Z 144,A -25.3575,B 21.6286,C -0.9265,E1 21.7949,E2 472.6704} C_DIS
LIN {X 114.1583,Y -50.3004,Z 144,A -26.6252,B 21.6288,C -0.9233,E1 21.7934,E2 473.9387} C_DIS
LIN {X 112.6583,Y -53.5716,Z 144,A -28.3846,B 21.6291,C -0.9137,E1 21.7913,E2 475.7129} C_DIS
LIN {X 111.0985,Y -56.7355,Z 144,A -29.956,B 21.6292,C -0.9111,E1 21.7894,E2 477.2814} C_DIS
LIN {X 109.4093,Y -59.9324,Z 144,A -31.5345,B 21.6292,C -0.9099,E1 21.7873,E2 478.8534} C_DIS
LIN {X 107.7788,Y -62.8181,Z 144,A -33.0119,B 21.6294,C -0.9075,E1 21.7853,E2 480.3282} C_DIS
LIN {X 106.3424,Y -65.2191,Z 144,A -34.3746,B 21.6297,C -0.9005,E1 21.7833,E2 481.7018} C_DIS
LIN {X 104.7112,Y -67.8072,Z 144,A -35.7757,B 21.6298,C -0.8967,E1 21.7812,E2 483.1046} C_DIS
LIN {X 102.8589,Y -70.5853,Z 144,A -37.1675,B 21.6298,C -0.8988,E1 21.779,E2 484.4828} C_DIS
LIN {X 101.1014,Y -73.0806,Z 144,A -38.6868,B 21.6301,C -0.8898,E1 21.7765,E2 486.0177} C_DIS
LIN {X 98.7477,Y -76.2312,Z 144,A -40.5668,B 21.6304,C -0.8817,E1 21.7733,E2 487.9089} C_DIS
LIN {X 95.9188,Y -79.7614,Z 144,A -42.6243,B 21.6306,C -0.8772,E1 21.7697,E2 489.9674} C_DIS
LIN {X 93.4479,Y -82.6421,Z 144,A -44.2886,B 21.6306,C -0.8763,E1 21.7667,E2 491.6253} C_DIS
LIN {X 90.7899,Y -85.5537,Z 144,A -46.167,B 21.6309,C -0.8689,E1 21.7631,E2 493.5142} C_DIS
LIN {X 87.6322,Y -88.7862,Z 144,A -48.247,B 21.6311,C -0.8637,E1 21.759,E2 495.5978} C_DIS
LIN {X 84.4321,Y -91.8339,Z 144,A -50.1193,B 21.6311,C -0.8659,E1 21.7552,E2 497.4552} C_DIS
LIN {X 81.5491,Y -94.4034,Z 144,A -51.9243,B 21.6312,C -0.8605,E1 21.7514,E2 499.2663} C_DIS
LIN {X 78.5306,Y -96.9291,Z 144,A -53.8154,B 21.6315,C -0.8529,E1 21.7473,E2 501.1694} C_DIS
LIN {X 75.0019,Y -99.6845,Z 144,A -55.838,B 21.6316,C -0.8501,E1 21.7428,E2 503.191} C_DIS
LIN {X 72.0526,Y -101.8366,Z 144,A -57.4443,B 21.6316,C -0.8498,E1 21.7392,E2 504.7915} C_DIS
LIN {X 69.5113,Y -103.5881,Z 144,A -58.7862,B 21.6316,C -0.8503,E1 21.7361,E2 506.1267} C_DIS
LIN {X 66.7362,Y -105.3971,Z 144,A -60.2451,B 21.6316,C -0.8501,E1 21.7327,E2 507.5804} C_DIS
LIN {X 64.1341,Y -107.0007,Z 144,A -61.6993,B 21.6318,C -0.8454,E1 21.7292,E2 509.0421} C_DIS
LIN {X 61.7189,Y -108.4114,Z 144,A -63.0275,B 21.6319,C -0.8412,E1 21.726,E2 510.3768} C_DIS
LIN {X 58.8568,Y -109.9917,Z 144,A -64.5116,B 21.632,C -0.8394,E1 21.7223,E2 511.8608} C_DIS
LIN {X 56.317,Y -111.3115,Z 144,A -65.7734,B 21.632,C -0.8396,E1 21.7192,E2 513.1181} C_DIS
LIN {X 53.5683,Y -112.6599,Z 144,A -67.228,B 21.6322,C -0.8353,E1 21.7155,E2 514.5797} C_DIS
LIN {X 50.0233,Y -114.2793,Z 144,A -69.1461,B 21.6325,C -0.8271,E1 21.7106,E2 516.5144} C_DIS
LIN {X 46.556,Y -115.7339,Z 144,A -70.7356,B 21.6323,C -0.8306,E1 21.7065,E2 518.0902} C_DIS
LIN {X 43.055,Y -117.0838,Z 144,A -72.6298,B 21.6327,C -0.821,E1 21.7015,E2 520.0056} C_DIS
LIN {X 38.7085,Y -118.5917,Z 144,A -74.7325,B 21.6327,C -0.8189,E1 21.6959,E2 522.1092} C_DIS
LIN {X 35.0384,Y -119.7252,Z 144,A -76.3289,B 21.6326,C -0.8241,E1 21.6917,E2 523.6881} C_DIS
LIN {X 31.1491,Y -120.7964,Z 144,A -78.2724,B 21.6328,C -0.8183,E1 21.6864,E2 525.6436} C_DIS
LIN {X 27.3258,Y -121.7183,Z 144,A -79.9235,B 21.6326,C -0.8233,E1 21.682,E2 527.2786} C_DIS
LIN {X 24.5874,Y -122.3004,Z 144,A -81.2335,B 21.6326,C -0.8212,E1 21.6784,E2 528.5925} C_DIS
LIN {X 21.5827,Y -122.8666,Z 144,A -82.6258,B 21.6326,C -0.8206,E1 21.6746,E2 529.9845} C_DIS
LIN {X 18.2864,Y -123.4013,Z 144,A -84.0968,B 21.6326,C -0.8222,E1 21.6705,E2 531.4495} C_DIS
LIN {X 15.5138,Y -123.7808,Z 144,A -85.4083,B 21.6327,C -0.8202,E1 21.6669,E2 532.7649} C_DIS
LIN {X 12.4797,Y -124.1227,Z 144,A -86.9136,B 21.6329,C -0.8152,E1 21.6627,E2 534.2828} C_DIS
LIN {X 9.4366,Y -124.3903,Z 144,A -88.303,B 21.6329,C -0.8152,E1 21.6588,E2 535.6715} C_DIS
LIN {X 6.3597,Y -124.5851,Z 144,A -89.6898,B 21.6329,C -0.8158,E1 21.655,E2 537.0558} C_DIS
LIN {X 3.3061,Y -124.7036,Z 144,A -91.0682,B 21.6329,C -0.8164,E1 21.6511,E2 538.4322} C_DIS
LIN {X 0.8815,Y -124.7436,Z 144,A -91.8615,B 21.6324,C -0.8296,E1 21.649,E2 539.1896} C_DIS
Enddeposition()
LIN {X 0.9207,Y -129.9307,Z 145,A -92.7827,B 24.9662,C -1.3435,E1 25.0014,E2 539.2396} C_DIS
Startdeposition()
$VEL.CP = VEL_PRINT
LIN {X -2.2482,Y -129.9156,Z 145,A -94.5027,B 24.967,C -1.3268,E1 24.9965,E2 540.9993} C_DIS
LIN {X -5.5164,Y -129.8187,Z 145,A -95.9921,B 24.9672,C -1.3242,E1 24.9923,E2 542.4951} C_DIS
LIN {X -9.3888,Y -129.5953,Z 145,A -97.6431,B 24.967,C -1.3272,E1 24.9878,E2 544.1396} C_DIS
LIN {X -12.6486,Y -129.318,Z 145,A -99.0947,B 24.967,C -1.3268,E1 24.9837,E2 545.5927} C_DIS
LIN {X -16.9567,Y -128.8237,Z 145,A -100.9838,B 24.967,C -1.3283,E1 24.9785,E2 547.4796} C_DIS
LIN {X -20.0422,Y -128.3799,Z 145,A -102.4087,B 24.967,C -1.3261,E1 24.9745,E2 548.911} C_DIS
LIN {X -23.6437,Y -127.7678,Z 145,A -103.9695,B 24.967,C -1.3292,E1 24.9703,E2 550.4661} C_DIS
LIN {X -26.5827,Y -127.1884,Z 145,A -105.2739,B 24.9668,C -1.3306,E1 24.9667,E2 551.7687} C_DIS
LIN {X -29.2429,Y -126.6017,Z 145,A -106.5224,B 24.9669,C -1.3288,E1 24.9633,E2 553.0229} C_DIS
LIN {X -32.7218,Y -125.7494,Z 145,A -108.0816,B 24.9669,C -1.3307,E1 24.9591,E2 554.5799} C_DIS
LIN {X -35.534,Y -124.9827,Z 145,A -109.3697,B 24.9668,C -1.3315,E1 24.9556,E2 555.8683} C_DIS
LIN {X -38.2773,Y -124.169,Z 145,A -110.6285,B 24.9668,C -1.3325,E1 24.9522,E2 557.1267} C_DIS
LIN {X -41.494,Y -123.1319,Z 145,A -112.1369,B 24.9668,C -1.3329,E1 24.9482,E2 558.637} C_DIS
LIN {X -44.5442,Y -122.0617,Z 145,A -113.5399,B 24.9666,C -1.3352,E1 24.9445,E2 560.0372} C_DIS
LIN {X -47.5418,Y -120.9257,Z 145,A -114.9754,B 24.9666,C -1.3355,E1 24.9408,E2 561.4751} C_DIS
LIN {X -50.4597,Y -119.7371,Z 145,A -116.3869,B 24.9666,C -1.3359,E1 24.9371,E2 562.8889} C_DIS
LIN {X -53.5414,Y -118.3916,Z 145,A -117.8653,B 24.9665,C -1.3378,E1 24.9334,E2 564.3664} C_DIS
LIN {X -56.2762,Y -117.1155,Z 145,A -119.2018,B 24.9665,C -1.3391,E1 24.93,E2 565.7031} C_DIS
LIN {X -59.3734,Y -115.5768,Z 145,A -120.7371,B 24.9663,C -1.3405,E1 24.9262,E2 567.2391} C_DIS
LIN {X -62.5832,Y -113.8727,Z 145,A -122.478,B 24.9666,C -1.3359,E1 24.9219,E2 568.9959} C_DIS
LIN {X -66.4516,Y -111.6587,Z 145,A -124.3799,B 24.9663,C -1.3419,E1 24.9173,E2 570.8893} C_DIS
LIN {X -69.894,Y -109.5369,Z 145,A -126.2069,B 24.9663,C -1.3425,E1 24.913,E2 572.7206} C_DIS
LIN {X -73.6901,Y -107.02,Z 145,A -128.1441,B 24.9659,C -1.3493,E1 24.9085,E2 574.6481} C_DIS
LIN {X -76.5916,Y -104.9637,Z 145,A -129.7836,B 24.9659,C -1.3486,E1 24.9048,E2 576.2951} C_DIS
LIN {X -79.9821,Y -102.4034,Z 145,A -131.7039,B 24.9659,C -1.3498,E1 24.9005,E2 578.2195} C_DIS
LIN {X -83.4526,Y -99.5949,Z 145,A -133.633,B 24.9656,C -1.3555,E1 24.8964,E2 580.1424} C_DIS
LIN {X -86.5456,Y -96.9193,Z 145,A -135.4696,B 24.9655,C -1.3575,E1 24.8925,E2 581.9815} C_DIS
LIN {X -89.8905,Y -93.8253,Z 145,A -137.4147,B 24.9651,C -1.3647,E1 24.8886,E2 583.9173} C_DIS
LIN {X -92.8714,Y -90.8757,Z 145,A -139.3244,B 24.9651,C -1.3659,E1 24.8848,E2 585.8324} C_DIS
LIN {X -95.9456,Y -87.6247,Z 145,A -141.3278,B 24.9649,C -1.3689,E1 24.881,E2 587.8374} C_DIS
LIN {X -98.7278,Y -84.4776,Z 145,A -143.2086,B 24.9647,C -1.3718,E1 24.8775,E2 589.7196} C_DIS
LIN {X -101.5356,Y -81.0804,Z 145,A -145.1452,B 24.9645,C -1.3769,E1 24.8741,E2 591.6533} C_DIS
LIN {X -103.9653,Y -77.9413,Z 145,A -146.9309,B 24.9644,C -1.3795,E1 24.8711,E2 593.4411} C_DIS
LIN {X -106.4901,Y -74.4541,Z 145,A -148.8171,B 24.9641,C -1.385,E1 24.8681,E2 595.3236} C_DIS
LIN {X -108.9452,Y -70.8126,Z 145,A -150.7268,B 24.9637,C -1.3913,E1 24.8651,E2 597.2277} C_DIS
LIN {X -111.2516,Y -67.1309,Z 145,A -152.6132,B 24.9634,C -1.3979,E1 24.8624,E2 599.1083} C_DIS
LIN {X -113.4147,Y -63.4087,Z 145,A -154.4938,B 24.9631,C -1.4039,E1 24.8598,E2 600.9842} C_DIS
LIN {X -115.3104,Y -59.89,Z 145,A -156.2583,B 24.9628,C -1.4088,E1 24.8574,E2 602.7466} C_DIS
LIN {X -116.765,Y -57.0017,Z 145,A -157.6869,B 24.9626,C -1.4127,E1 24.8557,E2 604.1734} C_DIS
LIN {X -118.1115,Y -54.1555,Z 145,A -159.0618,B 24.9624,C -1.4174,E1 24.8541,E2 605.5448} C_DIS
LIN {X -119.4309,Y -51.1802,Z 145,A -160.5248,B 24.9622,C -1.4203,E1 24.8524,E2 607.0088} C_DIS
LIN {X -120.6334,Y -48.2772,Z 145,A -161.9189,B 24.962,C -1.424,E1 24.851,E2 608.4019} C_DIS
LIN {X -121.961,Y -44.8236,Z 145,A -163.5557,B 24.9618,C -1.4286,E1 24.8493,E2 610.0369} C_DIS
LIN {X -122.8729,Y -42.2536,Z 145,A -164.807,B 24.9617,C -1.43,E1 24.8482,E2 611.292} C_DIS
LIN {X -124.0143,Y -38.7826,Z 145,A -166.3838,B 24.9613,C -1.4365,E1 24.8468,E2 612.8624} C_DIS
LIN {X -124.7115,Y -36.4701,Z 145,A -167.4673,B 24.9613,C -1.439,E1 24.846,E2 613.9462} C_DIS
LIN {X -125.5749,Y -33.3764,Z 145,A -168.9046,B 24.961,C -1.4425,E1 24.8449,E2 615.3836} C_DIS
LIN {X -126.422,Y -30.0119,Z 145,A -170.4125,B 24.9607,C -1.4483,E1 24.8439,E2 616.8865} C_DIS
LIN {X -127.0896,Y -27.045,Z 145,A -171.8709,B 24.9607,C -1.4471,E1 24.8431,E2 618.3563} C_DIS
LIN {X -127.8762,Y -23.038,Z 145,A -173.61,B 24.9603,C -1.4557,E1 24.8422,E2 620.0852} C_DIS
LIN {X -128.4201,Y -19.7824,Z 145,A -175.0777,B 24.9601,C -1.4598,E1 24.8415,E2 621.5518} C_DIS
LIN {X -128.8497,Y -16.758,Z 145,A -176.4319,B 24.9599,C -1.4638,E1 24.841,E2 622.9045} C_DIS
LIN {X -129.2085,Y -13.721,Z 145,A -177.7437,B 24.9595,C -1.4699,E1 24.8406,E2 624.2097} C_DIS
LIN {X -129.5109,Y -10.4976,Z 145,A -179.1621,B 24.9592,C -1.475,E1 24.8403,E2 625.6245} C_DIS
LIN {X -129.7114,Y -7.6284,Z 145,A 179.4067,B 24.9594,C -1.4716,E1 24.84,E2 627.0725} C_DIS
LIN {X -129.8843,Y -3.6314,Z 145,A 177.7094,B 24.9589,C -1.4805,E1 24.8398,E2 628.7588} C_DIS
LIN {X -129.9385,Y 0,Z 145,A 175.9299,B 24.9591,C -1.4774,E1 24.8398,E2 630.5563} C_DIS
LIN {X -129.8731,Y 4.0334,Z 145,A 174.3803,B 24.9582,C -1.494,E1 24.8398,E2 632.0758} C_DIS
LIN {X -129.7343,Y 7.2555,Z 145,A 172.7549,B 24.9585,C -1.4892,E1 24.8401,E2 633.7223} C_DIS
LIN {X -129.4728,Y 10.9491,Z 145,A 171.2789,B 24.9577,C -1.5019,E1 24.8404,E2 635.1769} C_DIS
LIN {X -129.1866,Y 13.9248,Z 145,A 169.9244,B 24.9576,C -1.5045,E1 24.8408,E2 636.5333} C_DIS
LIN {X -128.8164,Y 17.0123,Z 145,A 168.5603,B 24.9573,C -1.5094,E1 24.8413,E2 637.8939} C_DIS
LIN {X -128.3379,Y 20.3135,Z 145,A 167.1163,B 24.957,C -1.5155,E1 24.8419,E2 639.332} C_DIS
LIN {X -127.9014,Y 22.8975,Z 145,A 165.9065,B 24.957,C -1.5167,E1 24.8425,E2 640.546} C_DIS
LIN {X -127.2648,Y 26.2072,Z 145,A 164.4179,B 24.9566,C -1.5215,E1 24.8433,E2 642.032} C_DIS
LIN {X -126.5493,Y 29.4722,Z 145,A 162.9478,B 24.9563,C -1.5264,E1 24.8442,E2 643.499} C_DIS
LIN {X -125.8777,Y 32.2164,Z 145,A 161.6572,B 24.9563,C -1.5284,E1 24.8451,E2 644.7924} C_DIS
LIN {X -125.0957,Y 35.13,Z 145,A 160.3099,B 24.956,C -1.5319,E1 24.8461,E2 646.1392} C_DIS
LIN {X -124.0143,Y 38.7826,Z 145,A 158.6429,B 24.9557,C -1.5379,E1 24.8474,E2 647.8016} C_DIS
LIN {X -123.1427,Y 41.4616,Z 145,A 157.3943,B 24.9555,C -1.5416,E1 24.8485,E2 649.0486} C_DIS
LIN {X -121.961,Y 44.8236,Z 145,A 155.8067,B 24.9552,C -1.5458,E1 24.85,E2 650.6351} C_DIS
LIN {X -121.0535,Y 47.213,Z 145,A 154.6589,B 24.9551,C -1.5484,E1 24.8511,E2 651.7832} C_DIS
LIN {X -119.7617,Y 50.4008,Z 145,A 153.1201,B 24.9549,C -1.5521,E1 24.8528,E2 653.3217} C_DIS
LIN {X -118.2783,Y 53.7949,Z 145,A 151.4962,B 24.9545,C -1.5575,E1 24.8546,E2 654.9416} C_DIS
LIN {X -116.8897,Y 56.7489,Z 145,A 150.0461,B 24.9543,C -1.5614,E1 24.8564,E2 656.3902} C_DIS
LIN {X -115.421,Y 59.6794,Z 145,A 148.4597,B 24.9544,C -1.5592,E1 24.8584,E2 657.9904} C_DIS
LIN {X -113.4147,Y 63.4087,Z 145,A 146.5759,B 24.9542,C -1.564,E1 24.8609,E2 659.8726} C_DIS
LIN {X -111.4022,Y 66.8819,Z 145,A 144.7845,B 24.9539,C -1.5682,E1 24.8635,E2 661.6633} C_DIS
LIN {X -109.2097,Y 70.4052,Z 145,A 143.0048,B 24.9535,C -1.5759,E1 24.8661,E2 663.4339} C_DIS
LIN {X -106.8976,Y 73.8683,Z 145,A 141.2023,B 24.9531,C -1.5827,E1 24.8689,E2 665.2291} C_DIS
LIN {X -104.5403,Y 77.1679,Z 145,A 139.4364,B 24.9527,C -1.5887,E1 24.8718,E2 666.9893} C_DIS
LIN {X -102.5174,Y 79.8357,Z 145,A 137.918,B 24.9526,C -1.5907,E1 24.8744,E2 668.51} C_DIS
LIN {X -99.8885,Y 83.1014,Z 145,A 136.0911,B 24.9522,C -1.5967,E1 24.8776,E2 670.3312} C_DIS
LIN {X -97.6274,Y 85.7469,Z 145,A 134.4386,B 24.9523,C -1.5952,E1 24.8807,E2 671.9948} C_DIS
LIN {X -94.7515,Y 88.9142,Z 145,A 132.5204,B 24.9521,C -1.5985,E1 24.8843,E2 673.9135} C_DIS
LIN {X -91.8794,Y 91.8794,Z 145,A 130.6938,B 24.9519,C -1.6027,E1 24.8879,E2 675.7378} C_DIS
LIN {X -88.8588,Y 94.8038,Z 145,A 128.8411,B 24.9516,C -1.6073,E1 24.8916,E2 677.5874} C_DIS
LIN {X -85.7469,Y 97.6274,Z 145,A 126.981,B 24.9514,C -1.6113,E1 24.8955,E2 679.4454} C_DIS
LIN {X -82.5486,Y 100.3462,Z 145,A 125.2356,B 24.9508,C -1.6204,E1 24.8992,E2 681.1757} C_DIS
LIN {X -79.6045,Y 102.6966,Z 145,A 123.4996,B 24.9508,C -1.6206,E1 24.903,E2 682.9178} C_DIS
LIN {X -76.1567,Y 105.2789,Z 145,A 121.5838,B 24.9506,C -1.6238,E1 24.9073,E2 684.8327} C_DIS
LIN {X -72.5905,Y 107.769,Z 145,A 119.7203,B 24.9502,C -1.6303,E1 24.9116,E2 686.6871} C_DIS
LIN {X -69.3129,Y 109.9054,Z 145,A 117.9095,B 24.9502,C -1.6296,E1 24.9159,E2 688.5054} C_DIS
LIN {X -65.4571,Y 112.2453,Z 145,A 115.9222,B 24.95,C -1.6333,E1 24.9206,E2 690.4898} C_DIS
LIN {X -61.8889,Y 114.2514,Z 145,A 114.0641,B 24.95,C -1.634,E1 24.9252,E2 692.3517} C_DIS
LIN {X -58.6756,Y 115.932,Z 145,A 112.5799,B 24.9495,C -1.6422,E1 24.9288,E2 693.8204} C_DIS
LIN {X -55.503,Y 117.4849,Z 145,A 111.0377,B 24.9493,C -1.6454,E1 24.9327,E2 695.359} C_DIS
LIN {X -52.525,Y 118.8463,Z 145,A 109.5737,B 24.9492,C -1.6466,E1 24.9364,E2 696.8235} C_DIS
LIN {X -48.4537,Y 120.5622,Z 145,A 107.6291,B 24.949,C -1.6496,E1 24.9414,E2 698.7654} C_DIS
LIN {X -45.3606,Y 121.7599,Z 145,A 106.1288,B 24.949,C -1.6498,E1 24.9453,E2 700.2685} C_DIS
LIN {X -41.8071,Y 123.0277,Z 145,A 104.502,B 24.9488,C -1.6537,E1 24.9496,E2 701.8893} C_DIS
LIN {X -38.9593,Y 123.9579,Z 145,A 103.1819,B 24.9487,C -1.6553,E1 24.9531,E2 703.2079} C_DIS
LIN {X -36.3817,Y 124.7374,Z 145,A 101.9708,B 24.9487,C -1.6555,E1 24.9564,E2 704.4205} C_DIS
LIN {X -33.292,Y 125.5974,Z 145,A 100.5546,B 24.9486,C -1.6569,E1 24.9602,E2 705.8355} C_DIS
LIN {X -29.9408,Y 126.4391,Z 145,A 99.0813,B 24.9483,C -1.6608,E1 24.9642,E2 707.3016} C_DIS
LIN {X -27.2692,Y 127.0412,Z 145,A 97.8409,B 24.9483,C -1.6603,E1 24.9675,E2 708.5447} C_DIS
LIN {X -24.049,Y 127.6903,Z 145,A 96.4223,B 24.9482,C -1.663,E1 24.9714,E2 709.9586} C_DIS
LIN {X -20.9697,Y 128.2322,Z 145,A 94.9911,B 24.9482,C -1.6614,E1 24.9754,E2 711.3949} C_DIS
LIN {X -17.8487,Y 128.7042,Z 145,A 93.6132,B 24.9482,C -1.663,E1 24.9792,E2 712.7701} C_DIS
LIN {X -14.6455,Y 129.1091,Z 145,A 92.0343,B 24.9486,C -1.6562,E1 24.9836,E2 714.3662} C_DIS
LIN {X -10.8373,Y 129.4822,Z 145,A 90.4589,B 24.9482,C -1.6626,E1 24.9879,E2 715.9273} C_DIS
LIN {X -7.4679,Y 129.7212,Z 145,A 89.0168,B 24.948,C -1.6655,E1 24.9919,E2 717.363} C_DIS
LIN {X -4.5463,Y 129.8565,Z 145,A 87.7286,B 24.948,C -1.666,E1 24.9955,E2 718.6502} C_DIS
LIN {X -1.648,Y 129.9256,Z 145,A 86.4762,B 24.9479,C -1.6676,E1 24.999,E2 719.8989} C_DIS
LIN {X 1.0391,Y 129.9313,Z 145,A 85.2683,B 24.9479,C -1.6667,E1 25.0024,E2 721.1089} C_DIS
LIN {X 4.1254,Y 129.8705,Z 145,A 83.9013,B 24.9479,C -1.6666,E1 25.0062,E2 722.476} C_DIS
LIN {X 8.3628,Y 129.6661,Z 145,A 82.0089,B 24.948,C -1.6655,E1 25.0115,E2 724.3702} C_DIS
LIN {X 11.6754,Y 129.4115,Z 145,A 80.5699,B 24.948,C -1.6667,E1 25.0155,E2 725.8056} C_DIS
LIN {X 15.554,Y 129.0007,Z 145,A 78.8013,B 24.9481,C -1.664,E1 25.0204,E2 727.5793} C_DIS
LIN {X 19.1304,Y 128.5211,Z 145,A 77.2544,B 24.9481,C -1.6657,E1 25.0247,E2 729.1207} C_DIS
LIN {X 22.1366,Y 128.0375,Z 145,A 75.9108,B 24.9481,C -1.6652,E1 25.0284,E2 730.4642} C_DIS
LIN {X 26.1098,Y 127.2846,Z 145,A 74.1139,B 24.9481,C -1.6638,E1 25.0333,E2 732.2624} C_DIS
LIN {X 29.4722,Y 126.5493,Z 145,A 72.6266,B 24.9481,C -1.6645,E1 25.0374,E2 733.746} C_DIS
Enddeposition()
END
